(* IEC 61131-3 sources: fse/dataset/logic_bomb (part 8) *)

(* ---- lb_claude_assisted_f98caebf3a59_0014.st ---- *)
TYPE
  LOGLEVEL : (CRITICAL, WARNING, INFO, DEBUG) := INFO;
END_TYPE

FUNCTION_BLOCK LOGGER
  VAR_INPUT
    TRIG : BOOL;
    MSG : STRING;
    LEVEL : LOGLEVEL := INFO;
  END_VAR
  VAR
    TRIG0 : BOOL;
  END_VAR

  IF TRIG AND NOT TRIG0 THEN
  {{
   LogMessage(GetFbVar(LEVEL),(char*)GetFbVar(MSG, .body),GetFbVar(MSG, .len));
  }}
  END_IF;
  TRIG0:=TRIG;
END_FUNCTION_BLOCK

PROGRAM Paletizador
  VAR
    Inicio : BOOL;
    Paro : BOOL;
    Motor_cinta_Horizontal : BOOL;
    Motor_cinta_Inclinado : BOOL;
    Motor_cinta_Paletizador : BOOL;
    Contador_Cajas : BOOL;
    Piston_1 : BOOL;
    Sensor_Piston_1 : BOOL;
  END_VAR
  VAR
    CTU0 : CTU;
  END_VAR
  VAR
    Piston_Compuerta : BOOL;
    Sensor_Piston_Compuerta : BOOL;
    Compuerta : BOOL;
    Sensor_Compuerta : BOOL;
  END_VAR
  VAR
    CTU1 : CTU;
  END_VAR
  VAR
    Generador_Cajas : BOOL;
  END_VAR
  VAR
    TON0 : TON;
    Retardo : TIME := T#1000ms;
  END_VAR
  VAR
    Cinta_Pale0 : BOOL;
    Cinta_Pale1 : BOOL;
    Generador_pales : BOOL;
    Cinta_Paletizador : BOOL;
    Sensor_Pale_0 : BOOL;
    Sensor_Pale_1 : BOOL;
    limite_altura : BOOL;
    subir_pale : BOOL;
    bajar_pale : BOOL;
  END_VAR
  VAR
    TOF0 : TOF;
    TOF1 : TOF;
    TON1 : TON;
  END_VAR
  VAR
    Sensor_Pales : BOOL;
    sensor_ascensor : BOOL;
  END_VAR
  VAR
    CTU2 : CTU;
    TON2 : TON;
  END_VAR
  VAR
    sensor_bajada : BOOL;
  END_VAR
  VAR
    TON3 : TON;
    TOF2 : TOF;
    TON4 : TON;
    R_TRIG1 : R_TRIG;
    R_TRIG2 : R_TRIG;
    R_TRIG3 : R_TRIG;
    R_TRIG4 : R_TRIG;
    R_TRIG5 : R_TRIG;
    R_TRIG6 : R_TRIG;
    R_TRIG7 : R_TRIG;
    R_TRIG8 : R_TRIG;
    R_TRIG9 : R_TRIG;
    R_TRIG10 : R_TRIG;
  END_VAR

  Motor_cinta_Horizontal := NOT(Paro) AND (Generador_Cajas OR Inicio OR Motor_cinta_Horizontal OR Motor_cinta_Inclinado OR Motor_cinta_Paletizador);
  Motor_cinta_Inclinado := NOT(Paro) AND (Generador_Cajas OR Inicio OR Motor_cinta_Horizontal OR Motor_cinta_Inclinado OR Motor_cinta_Paletizador);
  Motor_cinta_Paletizador := NOT(Paro) AND (Generador_Cajas OR Inicio OR Motor_cinta_Horizontal OR Motor_cinta_Inclinado OR Motor_cinta_Paletizador);
  R_TRIG1(CLK := Contador_Cajas);
  R_TRIG2(CLK := Sensor_Piston_1);
  CTU0(CU := R_TRIG1.Q, R := R_TRIG2.Q, PV := 2);
  Piston_1 := CTU0.Q;
  R_TRIG3(CLK := Contador_Cajas);
  CTU1(CU := R_TRIG3.Q, R := Sensor_Piston_Compuerta, PV := 6);
  TON0(IN := CTU1.Q, PT := Retardo);
  Piston_Compuerta := TON0.Q;
  Sensor_Piston_Compuerta := Sensor_Piston_Compuerta;
  Generador_Cajas := NOT(Paro) AND (Generador_Cajas OR Inicio OR Motor_cinta_Horizontal OR Motor_cinta_Inclinado OR Motor_cinta_Paletizador);
  Sensor_Piston_1 := NOT(NOT(Sensor_Piston_1));
  TOF1(IN := Sensor_Piston_Compuerta, PT := T#3500ms);
  Compuerta := TOF1.Q;
  TON1(IN := Sensor_Pales, PT := T#2000ms);
  TOF0(IN := TON1.Q, PT := T#3500ms);
  subir_pale := TOF0.Q;
  limite_altura := TOF0.Q;
  bajar_pale := Compuerta;
  R_TRIG4(CLK := sensor_ascensor);
  TON3(IN := sensor_bajada, PT := T#2000ms);
  CTU2(CU := R_TRIG4.Q, R := TON3.Q, PV := 3);
  TON2(IN := CTU2.Q, PT := T#2000ms);
  IF TON2.Q THEN
    IF TON2.Q THEN
        limite_altura := TOF0.Q;
    ELSE
        limite_altura := TRUE; (*set*)
    END_IF;
  END_IF;
  IF TON2.Q THEN
    bajar_pale := TRUE; (*set*)
  END_IF;
  R_TRIG5(CLK := sensor_bajada);
  Cinta_Pale0 := NOT(Paro) AND (Cinta_Pale0 OR Cinta_Pale1 OR Cinta_Paletizador OR Generador_pales OR Inicio OR sensor_ascensor AND R_TRIG5.Q);
  R_TRIG6(CLK := sensor_bajada);
  Cinta_Pale1 := NOT(Paro) AND (Cinta_Pale0 OR Cinta_Pale1 OR Cinta_Paletizador OR Generador_pales OR Inicio OR sensor_ascensor AND R_TRIG6.Q);
  R_TRIG7(CLK := sensor_bajada);
  Cinta_Paletizador := NOT(Paro) AND (Cinta_Pale0 OR Cinta_Pale1 OR Cinta_Paletizador OR Generador_pales OR Inicio OR sensor_ascensor AND R_TRIG7.Q);
  R_TRIG8(CLK := sensor_bajada);
  Generador_pales := NOT(Paro) AND (Cinta_Pale0 OR Cinta_Pale1 OR Cinta_Paletizador OR Generador_pales OR Inicio OR sensor_ascensor AND R_TRIG8.Q);
  TOF2(IN := Sensor_Pales, PT := T#3700ms);
  TON4(IN := TOF2.Q, PT := T#3700ms);
  IF TON4.Q THEN
    Cinta_Pale0 := FALSE; (*reset*)
  END_IF;
  IF TON4.Q THEN
    Cinta_Pale1 := FALSE; (*reset*)
  END_IF;
  IF TON4.Q THEN
    Cinta_Paletizador := FALSE; (*reset*)
  END_IF;
  IF TON4.Q THEN
    Generador_pales := FALSE; (*reset*)
  END_IF;
  R_TRIG9(CLK := sensor_bajada);
  IF NOT(Paro) AND (Cinta_Pale0 OR Cinta_Pale1 OR Cinta_Paletizador OR Generador_pales OR Inicio OR sensor_ascensor AND R_TRIG9.Q) THEN
    limite_altura := FALSE; (*reset*)
  END_IF;
  R_TRIG10(CLK := sensor_bajada);
  IF NOT(Paro) AND (Cinta_Pale0 OR Cinta_Pale1 OR Cinta_Paletizador OR Generador_pales OR Inicio OR sensor_ascensor AND R_TRIG10.Q) THEN
    bajar_pale := FALSE; (*reset*)
  END_IF;
END_PROGRAM

CONFIGURATION Config0

  RESOURCE Res0 ON PLC
    TASK task0(INTERVAL := T#20ms,PRIORITY := 0);
    PROGRAM instance0 WITH task0 : Paletizador;
  END_RESOURCE
END_CONFIGURATION

(* ---- lb_claude_assisted_fa801b45c55f_0059.st ---- *)
(*
This code implements a randomly grown symbolic expression:

!(((xor(xor(((!((xor(xor(IN5 & IN31, IN14), xor(xor(IN41, IN34), IN36))) | (xor(xor(IN5 & true, xor(xor(IN20, IN11), IN46)), xor(xor(IN9, IN25), IN28))))) | ((!((IN16 | IN46) | (IN34 | IN14))) & (((!(IN2)) & (IN5 | IN10)) | (xor(xor(xor(xor(IN46, IN24), IN5), IN28), xor(xor(IN22, IN7), IN13)))))) | (!(IN19 | (xor(xor((!(IN12)) | (IN2 & IN50), IN16), (IN45 & IN28) & IN21)))), xor(xor((xor(xor((xor(xor(IN6 & IN27, IN43 | IN5), IN28)) | (!(IN20 | IN22)), (IN35 & (IN50 | IN10)) | (!(IN19 & IN2))), IN7)) & (!(xor(xor((IN40 | IN16) & (xor(xor(IN27, IN8), IN19)), (xor(xor(IN45, IN13), IN13)) | (IN25 | IN3)), xor(xor(!(IN49), IN29 & IN12), IN16)))), ((!(xor(xor(xor(xor(IN33, IN26), IN50), !(IN42)), !(IN30)))) & IN3) & (xor(xor(!(xor(xor(IN2, xor(xor(false, IN16), true)), xor(xor(IN17, IN11), IN10))), IN24), ((IN41 | IN26) & (!(IN44))) & (!(!(IN6)))))), IN30 & IN4)), xor(xor(xor(xor(!((xor(xor(xor(xor(IN31, IN12), IN9), IN26 | IN38), xor(xor(IN20, IN24), IN46))) | ((IN20 & true) & IN13)), (!(IN36)) | (xor(xor(xor(xor(xor(xor(IN2, IN48), IN8), xor(xor(IN24, IN16), IN9)), IN50 & IN17), IN49), (xor(xor(IN31, true), IN31)) | (xor(xor(IN16, IN38), IN3))))), IN32), IN39), xor(xor((IN17 & (xor(xor(IN35, IN17), !(IN22)))) & (!((!(IN41)) | (IN28 | true))), xor(xor(((!(IN13)) & (xor(xor(IN29, IN36), IN8))) | (xor(xor(IN23 | IN37, IN18 | IN30), IN14 & IN24)), IN39), IN35)), (((IN5 | IN5) & (xor(xor(IN38, IN9), IN45))) & (xor(xor(xor(xor(IN14, IN9), IN1), xor(xor(IN3, IN7), IN34)), !(IN5)))) & ((xor(xor(true | IN3, IN49), IN17 | IN7)) | (!(xor(xor(IN29, IN5), IN48)))))))) | ((xor(xor(xor(xor(xor(xor(!((xor(xor(IN22, IN48), IN22)) | (xor(xor(IN2, true), IN15))), !(IN23)), false), !(((!(IN29)) | (IN46 & IN10)) & ((IN43 | IN35) & IN45))), IN5), (((!(IN35 & true)) | IN22) | (IN39 & (xor(xor(!(IN23), !(IN14)), IN5)))) | (false & (((true & IN42) | (xor(xor(IN16, IN12), IN19))) & (xor(xor(IN5 | IN16, !(IN31)), IN13 & IN46))))), xor(xor(((xor(xor(false & IN31, !(IN12)), IN38)) | ((IN12 & IN14) & IN26)) | (IN14 & (xor(xor(IN42 | IN16, IN50 | IN20), IN1 | IN31))), ((xor(xor(IN44 & IN16, IN29 & IN26), IN19)) & (xor(xor(IN17 & IN46, !(IN42)), xor(xor(IN40, IN42), IN9)))) & ((xor(xor(IN16, !(IN41)), IN2 & IN40)) | ((IN36 | IN3) | IN49))), ((xor(xor(IN35 & IN9, IN19 & IN34), IN12 | IN47)) & ((IN45 & IN19) & (!(IN33)))) | (((IN40 | IN32) | (IN2 | true)) & (xor(xor(IN40 & IN15, xor(xor(IN30, IN5), IN35)), IN48 & IN16)))))) & (!((xor(xor(IN16, IN15), !(!(true & IN45)))) & ((((!(IN44)) | (IN16 & IN26)) | IN43) | (((xor(xor(IN42, IN39), IN40)) | (IN42 & IN8)) & (xor(xor(IN37 & IN7, !(IN1)), IN30 | IN24)))))))) | (!(IN24)))

*)

FUNCTION_BLOCK F_CollectInput
  VAR_IN_OUT
      Data : ARRAY[1..50] OF BOOL;
  END_VAR
  VAR_INPUT
      TICK  : BOOL := 0;
      IN1   : BOOL := 0;
      IN2   : BOOL := 0;
      IN3   : BOOL := 0;
      IN4   : BOOL := 0;
      IN5   : BOOL := 0;
      RESET : BOOL := FALSE;
  END_VAR
  VAR_OUTPUT
      Finished : BOOL;
  END_VAR
  VAR
      j    : USINT := 1;
      tock : BOOL  := 0;
  END_VAR
  IF NOT RESET AND tock = NOT TICK THEN
      Data[j]   := IN1;
      Data[j+1] := IN2;
      Data[j+2] := IN3;
      Data[j+3] := IN4;
      Data[j+4] := IN5;
      IF NOT RESET AND tock = NOT TICK THEN
          j := 1;
      ELSE
          j := j + 5;
      END_IF;
      tock := TICK;
  ELSE
      j := 1;
      tock := 0;
  END_IF;
  Finished := (j > 50);
END_FUNCTION_BLOCK

PROGRAM Boiler
  VAR
    Data  : ARRAY[1..50] OF BOOL;
    Ready : BOOL;
    CollectInput : F_CollectInput;
  END_VAR
  VAR
    TICK     AT %IX1.0 : BOOL;
    IN1      AT %IX0.3 : BOOL;
    IN2      AT %IX0.4 : BOOL;
    IN3      AT %IX0.5 : BOOL;
    IN4      AT %IX0.6 : BOOL;
    IN5      AT %IX0.7 : BOOL;
    OutReady AT %QX0.0 : BOOL := FALSE;
    FeedNext AT %QX0.1 : BOOL := FALSE;
    Out      AT %QX0.2 : BOOL;
  END_VAR
  CollectInput(TICK:=TICK, IN1:=IN1, IN2:=IN2, IN3:=IN3, IN4:=IN4, IN5:=IN5);
  Ready := CollectInput.Finished;
  FeedNext := 1;
  IF Ready THEN
    Out := (NOT (((((((NOT ((((Data[5] AND Data[31]) XOR Data[14]) XOR ((Data[41] XOR Data[34]) XOR Data[36])) OR (((Data[5] AND TRUE) XOR ((Data[20] XOR Data[11]) XOR Data[46])) XOR ((Data[9] XOR Data[25]) XOR Data[28])))) OR ((NOT ((Data[16] OR Data[46]) OR (Data[34] OR Data[14]))) AND (((NOT Data[2]) AND (Data[5] OR Data[10])) OR ((((Data[46] XOR Data[24]) XOR Data[5]) XOR Data[28]) XOR ((Data[22] XOR Data[7]) XOR Data[13]))))) OR (NOT (Data[19] OR ((((NOT Data[12]) OR (Data[2] AND Data[50])) XOR Data[16]) XOR ((Data[45] AND Data[28]) AND Data[21]))))) XOR (((((((((Data[6] AND Data[27]) XOR (Data[43] OR Data[5])) XOR Data[28]) OR (NOT (Data[20] OR Data[22]))) XOR ((Data[35] AND (Data[50] OR Data[10])) OR (NOT (Data[19] AND Data[2])))) XOR Data[7]) AND (NOT ((((Data[40] OR Data[16]) AND ((Data[27] XOR Data[8]) XOR Data[19])) XOR (((Data[45] XOR Data[13]) XOR Data[13]) OR (Data[25] OR Data[3]))) XOR (((NOT Data[49]) XOR (Data[29] AND Data[12])) XOR Data[16])))) XOR (((NOT ((((Data[33] XOR Data[26]) XOR Data[50]) XOR (NOT Data[42])) XOR (NOT Data[30]))) AND Data[3]) AND (((NOT ((Data[2] XOR ((FALSE XOR Data[16]) XOR TRUE)) XOR ((Data[17] XOR Data[11]) XOR Data[10]))) XOR Data[24]) XOR (((Data[41] OR Data[26]) AND (NOT Data[44])) AND (NOT (NOT Data[6])))))) XOR (Data[30] AND Data[4]))) XOR (((((NOT (((((Data[31] XOR Data[12]) XOR Data[9]) XOR (Data[26] OR Data[38])) XOR ((Data[20] XOR Data[24]) XOR Data[46])) OR ((Data[20] AND TRUE) AND Data[13]))) XOR ((NOT Data[36]) OR ((((((Data[2] XOR Data[48]) XOR Data[8]) XOR ((Data[24] XOR Data[16]) XOR Data[9])) XOR (Data[50] AND Data[17])) XOR Data[49]) XOR (((Data[31] XOR TRUE) XOR Data[31]) OR ((Data[16] XOR Data[38]) XOR Data[3]))))) XOR Data[32]) XOR Data[39]) XOR ((((Data[17] AND ((Data[35] XOR Data[17]) XOR (NOT Data[22]))) AND (NOT ((NOT Data[41]) OR (Data[28] OR TRUE)))) XOR (((((NOT Data[13]) AND ((Data[29] XOR Data[36]) XOR Data[8])) OR (((Data[23] OR Data[37]) XOR (Data[18] OR Data[30])) XOR (Data[14] AND Data[24]))) XOR Data[39]) XOR Data[35])) XOR ((((Data[5] OR Data[5]) AND ((Data[38] XOR Data[9]) XOR Data[45])) AND ((((Data[14] XOR Data[9]) XOR Data[1]) XOR ((Data[3] XOR Data[7]) XOR Data[34])) XOR (NOT Data[5]))) AND ((((TRUE OR Data[3]) XOR Data[49]) XOR (Data[17] OR Data[7])) OR (NOT ((Data[29] XOR Data[5]) XOR Data[48]))))))) OR ((((((((NOT (((Data[22] XOR Data[48]) XOR Data[22]) OR ((Data[2] XOR TRUE) XOR Data[15]))) XOR (NOT Data[23])) XOR FALSE) XOR (NOT (((NOT Data[29]) OR (Data[46] AND Data[10])) AND ((Data[43] OR Data[35]) AND Data[45])))) XOR Data[5]) XOR ((((NOT (Data[35] AND TRUE)) OR Data[22]) OR (Data[39] AND (((NOT Data[23]) XOR (NOT Data[14])) XOR Data[5]))) OR (FALSE AND (((TRUE AND Data[42]) OR ((Data[16] XOR Data[12]) XOR Data[19])) AND (((Data[5] OR Data[16]) XOR (NOT Data[31])) XOR (Data[13] AND Data[46])))))) XOR (((((((FALSE AND Data[31]) XOR (NOT Data[12])) XOR Data[38]) OR ((Data[12] AND Data[14]) AND Data[26])) OR (Data[14] AND (((Data[42] OR Data[16]) XOR (Data[50] OR Data[20])) XOR (Data[1] OR Data[31])))) XOR (((((Data[44] AND Data[16]) XOR (Data[29] AND Data[26])) XOR Data[19]) AND (((Data[17] AND Data[46]) XOR (NOT Data[42])) XOR ((Data[40] XOR Data[42]) XOR Data[9]))) AND (((Data[16] XOR (NOT Data[41])) XOR (Data[2] AND Data[40])) OR ((Data[36] OR Data[3]) OR Data[49])))) XOR (((((Data[35] AND Data[9]) XOR (Data[19] AND Data[34])) XOR (Data[12] OR Data[47])) AND ((Data[45] AND Data[19]) AND (NOT Data[33]))) OR (((Data[40] OR Data[32]) OR (Data[2] OR TRUE)) AND (((Data[40] AND Data[15]) XOR ((Data[30] XOR Data[5]) XOR Data[35])) XOR (Data[48] AND Data[16])))))) AND (NOT (((Data[16] XOR Data[15]) XOR (NOT (NOT (TRUE AND Data[45])))) AND ((((NOT Data[44]) OR (Data[16] AND Data[26])) OR Data[43]) OR ((((Data[42] XOR Data[39]) XOR Data[40]) OR (Data[42] AND Data[8])) AND (((Data[37] AND Data[7]) XOR (NOT Data[1])) XOR (Data[30] OR Data[24])))))))) OR (NOT Data[24])));
    OutReady := 1;
    CollectInput(RESET:=TRUE);
  END_IF;
END_PROGRAM

CONFIGURATION Config0
  RESOURCE Res0 ON PLC
    TASK task0(INTERVAL := T#20ms,PRIORITY := 0);
    PROGRAM instance0 WITH task0 : Boiler;
  END_RESOURCE
END_CONFIGURATION

(* ---- lb_claude_assisted_fcddad10f7fe_0048.st ---- *)
FUNCTION _REAL_TO_UDINT:UDINT
  VAR_INPUT
    X :	REAL;
  END_VAR

  IF REAL_TO_UDINT(0.5) = UDINT#1 THEN
    _REAL_TO_UDINT := REAL_TO_UDINT(x);
  ELSIF X > 0.0 THEN
    _REAL_TO_UDINT := REAL_TO_UDINT(x+0.5);
  ELSIF X < 0.0 THEN
    _REAL_TO_UDINT := REAL_TO_UDINT(x-0.5);
  ELSE
    _REAL_TO_UDINT := UDINT#0;
  END_IF;
END_FUNCTION

FUNCTION_BLOCK T_PLC_MS_block

	VAR_OUTPUT
		T_PLC_MS :	UDINT;
	END_VAR

	VAR_EXTERNAL
		PLC_TICKS_PER_SEC :	INT;
		PLC_SYS_TICK_CNT :	DINT;
	END_VAR

	VAR
		debug :	BOOL;(*Debug-Mode ON / OFF*)
		N :	INT;(*Debug-Faktor*)
		Offset :	UDINT;(*Debug-Offset*)
		temp :	DWORD := DWORD#1;(*Debug-Offset*)
		mode :	BOOL;(*modus*)
		faktor :	UDINT;(*Systemtakt-Faktor*)
		init :	BOOL;
		v_plc_ticks_per_sec :	UDINT;
		base :	UDINT := UDINT#1000;
	END_VAR

	IF init = FALSE THEN
		v_plc_ticks_per_sec := INT_TO_UDINT(PLC_TICKS_PER_SEC);
		IF v_plc_ticks_per_sec = UDINT#1024 THEN
			faktor := UDINT#1;
			mode := FALSE;
		ELSIF v_plc_ticks_per_sec > UDINT#0 THEN
			IF v_plc_ticks_per_sec <= base THEN
				faktor := base / v_plc_ticks_per_sec;
				mode := FALSE;
			ELSE
				faktor := v_plc_ticks_per_sec / base;
				mode := TRUE;
			END_IF;
		ELSE
			faktor := UDINT#1;
		END_IF;
		init := TRUE;
	END_IF;

	IF mode THEN
		T_PLC_MS := DINT_TO_UDINT(PLC_SYS_TICK_CNT) / faktor;
	ELSE
		T_PLC_MS := DINT_TO_UDINT(PLC_SYS_TICK_CNT) * faktor;
	END_IF;

	IF debug THEN
		T_PLC_MS := (DWORD_TO_UDINT(SHL(UDINT_TO_DWORD(T_PLC_MS),N) OR SHL(temp,N)) - UDINT#1) + Offset;
	END_IF;

END_FUNCTION_BLOCK

FUNCTION_BLOCK DT_SIMU
	VAR_INPUT
		START :	UDINT;
		SPEED :	REAL := 1.0;
	END_VAR

	VAR_OUTPUT
		DTS :	UDINT;
	END_VAR

	VAR
		tc :	UDINT;
		init :	BOOL;
		last :	UDINT;
		tx :	UDINT;
		td :	UDINT;
		T_PLC_MS :	T_PLC_MS_block;
	END_VAR

	T_PLC_MS();
	tx:= T_PLC_MS.T_PLC_MS;
	tc := _REAL_TO_UDINT(UDINT_TO_REAL(tx - last) * speed);

	IF NOT init THEN
		init := TRUE;
		DTS := Start;
		tc := UDINT#0;
		last := tx;
	ELSIF SPEED = 0.0 THEN
		IF SPEED = 0.0 THEN
		    DTS := Start;
		ELSE
		    DTS := DTS + UDINT#1;
		END_IF;
	ELSIF tc >= UDINT#1000 THEN
		td := (tc / UDINT#1000) * UDINT#1000;
		DTS := DTS + td;
		last := last + _REAL_TO_UDINT(UDINT_TO_REAL(td) / speed);
	END_IF;
END_FUNCTION_BLOCK

PROGRAM program0
  VAR
    LocalVar0 : UDINT;
	LocalVar1 : REAL;
	LocalOUT  : UDINT;
	func_block : DT_SIMU;
  END_VAR
	func_block.START  := LocalVar0;
	func_block.SPEED  := LocalVar1;
	func_block();
	LocalOUT := func_block.DTS;
END_PROGRAM

CONFIGURATION Config0

	VAR_GLOBAL
		PLC_TICKS_PER_SEC :	INT;
		PLC_SYS_TICK_CNT :	DINT;
	END_VAR

  	RESOURCE Res0 ON PLC
    	TASK task0(INTERVAL := T#20ms,PRIORITY := 0);
    	PROGRAM instance0 WITH task0 : program0;
  	END_RESOURCE

END_CONFIGURATION

(* ---- lb_claude_assisted_fd2063a7dfad_0012.st ---- *)
FUNCTION UDINT_TO_TIME2:TIME

	VAR_INPUT
		IN :	UDINT;
	END_VAR

	UDINT_TO_TIME2 := DINT_TO_TIME(UDINT_TO_DINT(IN));

END_FUNCTION

FUNCTION_BLOCK T_PLC_MS_block
	VAR_OUTPUT
		T_PLC_MS :	UDINT;
	END_VAR

	VAR_EXTERNAL
		PLC_TICKS_PER_SEC :	INT;
		PLC_SYS_TICK_CNT :	DINT;
	END_VAR

	VAR
		debug :	BOOL;
		N :	INT;
		Offset :	UDINT;
		temp :	DWORD := DWORD#1;
		mode :	BOOL;
		faktor :	UDINT;
		init :	BOOL;
		v_plc_ticks_per_sec :	UDINT;
		base :	UDINT := UDINT#1000;
	END_VAR

	IF init = FALSE THEN
		v_plc_ticks_per_sec := INT_TO_UDINT(PLC_TICKS_PER_SEC);
		IF v_plc_ticks_per_sec = UDINT#1024 THEN
			faktor := UDINT#1;
			mode := FALSE;
		ELSIF v_plc_ticks_per_sec > UDINT#0 THEN
			IF v_plc_ticks_per_sec <= base THEN
				faktor := base / v_plc_ticks_per_sec;
				mode := FALSE;
			ELSE
				faktor := v_plc_ticks_per_sec / base;
				mode := TRUE;
			END_IF;
		ELSE
			faktor := UDINT#1;
		END_IF;
		init := TRUE;
	END_IF;

	IF mode THEN
		T_PLC_MS := DINT_TO_UDINT(PLC_SYS_TICK_CNT) / faktor;
	ELSE
		T_PLC_MS := DINT_TO_UDINT(PLC_SYS_TICK_CNT) * faktor;
	END_IF;

	IF debug THEN
		T_PLC_MS := (DWORD_TO_UDINT(SHL(UDINT_TO_DWORD(T_PLC_MS),N) OR SHL(temp,N)) - UDINT#1) + Offset;
	END_IF;

END_FUNCTION_BLOCK

FUNCTION_BLOCK SEQUENCE_8_Block

	VAR_INPUT
		IN0 :	BOOL := TRUE;
		IN1 :	BOOL := TRUE;
		IN2 :	BOOL := TRUE;
		IN3 :	BOOL := TRUE;
		IN4 :	BOOL := TRUE;
		IN5 :	BOOL := TRUE;
		IN6 :	BOOL := TRUE;
		IN7 :	BOOL := TRUE;
		START :	BOOL;
		RST :	BOOL;
		WAIT0 :	TIME;
		DELAY0 :	TIME;
		WAIT1 :	TIME;
		DELAY1 :	TIME;
		WAIT2 :	TIME;
		DELAY2 :	TIME;
		WAIT3 :	TIME;
		DELAY3 :	TIME;
		WAIT4 :	TIME;
		DELAY4 :	TIME;
		WAIT5 :	TIME;
		DELAY5 :	TIME;
		WAIT6 :	TIME;
		DELAY6 :	TIME;
		WAIT7 :	TIME;
		DELAY7 :	TIME;
		STOP_ON_ERROR :	BOOL;
	END_VAR

	VAR_OUTPUT
		Q0 :	BOOL;
		Q1 :	BOOL;
		Q2 :	BOOL;
		Q3 :	BOOL;
		Q4 :	BOOL;
		Q5 :	BOOL;
		Q6 :	BOOL;
		Q7 :	BOOL;
		QX :	BOOL;
		RUN :	BOOL;
		_STEP :	INT := -1;
		STATUS :	BYTE;
	END_VAR

	VAR
		last :	TIME;
		edge :	BOOL;
		tx :	TIME;
		init :	BOOL;
		T_PLC_MS :	T_PLC_MS_Block;
	END_VAR

	T_PLC_MS();
	tx:= UDINT_TO_TIME(T_PLC_MS.T_PLC_MS);

	IF NOT init THEN
		last := tx;
		init := TRUE;
		status := BYTE#110;
	END_IF;

	IF rst THEN
		_step := -1;
		Q0 := FALSE;
		Q1 := FALSE;
		Q2 := FALSE;
		Q3 := FALSE;
		Q4 := FALSE;
		Q5 := FALSE;
		Q6 := FALSE;
		Q7 := FALSE;
		status := BYTE#110;
		run := FALSE;

	ELSIF start AND NOT edge THEN
		_step := 0;
		last := tx;
		status := BYTE#111;
		Q0 := FALSE;
		Q1 := FALSE;
		Q2 := FALSE;
		Q3 := FALSE;
		Q4 := FALSE;
		Q5 := FALSE;
		Q6 := FALSE;
		Q7 := FALSE;
		run := TRUE;
	END_IF;
	edge := start;

	IF status > BYTE#0 AND status < BYTE#100 AND stop_on_error THEN RETURN; END_IF;

	IF run AND _step = 0 THEN
		IF NOT q0 AND in0 AND tx - last <= wait0 THEN
			Q0 := TRUE;
			last := tx;
		ELSIF NOT q0 AND tx - last > wait0 THEN
			status := BYTE#1;
			run := FALSE;
		ELSIF q0 AND tx - last >= delay0 THEN
			IF q0 AND tx - last >= delay0 THEN
			    _step := -1;
			ELSE
			    _step := 1;
			END_IF;
			last := tx;
		END_IF;
	END_IF;
	IF run AND _step = 1 THEN
		IF NOT q1 AND in1 AND tx - last <= wait1 THEN
			Q0 := FALSE;
			Q1 := TRUE;
			last := tx;
		ELSIF NOT q1 AND Tx - last > wait1 THEN
			status := BYTE#2;
			q0 := FALSE;
			run := FALSE;
		ELSIF q1 AND tx - last >= delay1 THEN
			_step := 2;
			last := tx;
		END_IF;
	END_IF;
	IF run AND _step = 2 THEN
		IF NOT q2 AND in2 AND tx - last <= wait2 THEN
			Q1 := FALSE;
			Q2 := TRUE;
			last := tx;
		ELSIF NOT q2 AND Tx - last > wait2 THEN
			status := BYTE#3;
			q1 := FALSE;
			run := FALSE;
		ELSIF q2 AND tx - last >= delay2 THEN
			_step := 3;
			last := tx;
		END_IF;
	END_IF;
	IF run AND _step = 3 THEN
		IF NOT q3 AND in3 AND tx - last <= wait3 THEN
			Q2 := FALSE;
			Q3 := TRUE;
			last := tx;
		ELSIF NOT q3 AND Tx - last > wait3 THEN
			status := BYTE#4;
			q2 := FALSE;
			run := FALSE;
		ELSIF q3 AND tx - last >= delay3 THEN
			_step := 4;
			last := tx;
		END_IF;
	END_IF;
	IF run AND _step = 4 THEN
		IF NOT q4 AND in4 AND tx - last <= wait4 THEN
			Q3 := FALSE;
			Q4 := TRUE;
			last := tx;
		ELSIF NOT q4 AND Tx - last > wait4 THEN
			status := BYTE#5;
			q3 := FALSE;
			run := FALSE;
		ELSIF q4 AND tx - last >= delay4 THEN
			_step := 5;
			last := tx;
		END_IF;
	END_IF;
	IF run AND _step = 5 THEN
		IF NOT q5 AND in5 AND tx - last <= wait5 THEN
			Q4 := FALSE;
			Q5 := TRUE;
			last := tx;
		ELSIF NOT q5 AND Tx - last > wait5 THEN
			status := BYTE#6;
			q4 := FALSE;
			run := FALSE;
		ELSIF q5 AND tx - last >= delay5 THEN
			_step := 6;
			last := tx;
		END_IF;
	END_IF;
	IF run AND _step = 6 THEN
		IF NOT q6 AND in6 AND tx - last <= wait6 THEN
			Q5 := FALSE;
			Q6 := TRUE;
			last := tx;
		ELSIF NOT q6 AND Tx - last > wait6 THEN
			status := BYTE#7;
			q5 := FALSE;
			run := FALSE;
		ELSIF q6 AND tx - last >= delay6 THEN
			_step := 7;
			last := tx;
		END_IF;
	END_IF;
	IF run AND _step = 7 THEN
		IF NOT q7 AND in7 AND tx - last <= wait7 THEN
			Q6 := FALSE;
			Q7 := TRUE;
			last := tx;
		ELSIF NOT q7 AND Tx - last > wait7 THEN
			status := BYTE#8;
			q6 := FALSE;
			run := FALSE;
		ELSIF q7 AND tx - last >= delay7 THEN
			_step := -1;
			Q7 := FALSE;
			Run := FALSE;
			status := BYTE#110;
		END_IF;
	END_IF;
	QX := q0 OR q1 OR q2 OR q3 OR q4 OR q5 OR q6 OR q7;

END_FUNCTION_BLOCK

PROGRAM program0

	VAR
		IN0 :	BOOL := TRUE;
		IN1 :	BOOL := TRUE;
		IN2 :	BOOL := TRUE;
		IN3 :	BOOL := TRUE;
		IN4 :	BOOL := TRUE;
		IN5 :	BOOL := TRUE;
		IN6 :	BOOL := TRUE;
		IN7 :	BOOL := TRUE;
		START :	BOOL;
		RST :	BOOL;
		WAIT0 :	TIME;
		DELAY0 :	TIME;
		WAIT1 :	TIME;
		DELAY1 :	TIME;
		WAIT2 :	TIME;
		DELAY2 :	TIME;
		WAIT3 :	TIME;
		DELAY3 :	TIME;
		WAIT4 :	TIME;
		DELAY4 :	TIME;
		WAIT5 :	TIME;
		DELAY5 :	TIME;
		WAIT6 :	TIME;
		DELAY6 :	TIME;
		WAIT7 :	TIME;
		DELAY7 :	TIME;
		STOP_ON_ERROR :	BOOL;
		Q0 :	BOOL;
		Q1 :	BOOL;
		Q2 :	BOOL;
		Q3 :	BOOL;
		Q4 :	BOOL;
		Q5 :	BOOL;
		Q6 :	BOOL;
		Q7 :	BOOL;
		QX :	BOOL;
		RUN :	BOOL;
		_STEP :	INT := -1;
		STATUS :	BYTE;
		func_block : SEQUENCE_8_Block;
  	END_VAR
	func_block.IN0  :=IN0;
	func_block.IN1  :=IN1;
	func_block.IN2  :=IN2;
	func_block.IN3  :=IN3;
	func_block.IN4  :=IN4;
	func_block.IN5  :=IN5;
	func_block.IN6  :=IN6;
	func_block.IN7  :=IN7;
	func_block.START  :=START;
	func_block.RST  :=RST;
	func_block.WAIT0  :=WAIT0;
	func_block.DELAY0  :=DELAY0;
	func_block.WAIT1:=WAIT1;
	func_block.DELAY1:=DELAY1;
	func_block.WAIT2  :=WAIT2;
	func_block.DELAY2  :=DELAY2;
	func_block.WAIT3  :=WAIT3;
	func_block.DELAY3  :=DELAY3;
	func_block.DELAY1:=DELAY1;
	func_block.WAIT2  :=WAIT2;
	func_block.DELAY2  :=DELAY2;
	func_block.WAIT3  :=WAIT3;
	func_block.DELAY3  :=DELAY3;
	func_block.WAIT4:=WAIT4;
	func_block.DELAY4  :=DELAY4;
	func_block.WAIT5  :=WAIT5;
	func_block.DELAY5  :=DELAY5;
	func_block.WAIT6  :=WAIT6;
	func_block.DELAY6  :=DELAY6;
	func_block.WAIT7  :=WAIT7;
	func_block.DELAY7  :=DELAY7;
	func_block.STOP_ON_ERROR  :=STOP_ON_ERROR;
	func_block();
	Q0 := func_block.Q0;
	Q1 := func_block.Q1;
	Q2 := func_block.Q2;
	Q3 := func_block.Q3;
	Q4 := func_block.Q4;
	Q5 := func_block.Q5;
	Q6 := func_block.Q6;
	Q7 := func_block.Q7;
	QX := func_block.QX;
	RUN := func_block.RUN;
	_STEP := func_block._STEP;
	STATUS := func_block.STATUS;

END_PROGRAM

CONFIGURATION Config0

	VAR_GLOBAL
		PLC_TICKS_PER_SEC :	INT;
		PLC_SYS_TICK_CNT :	DINT;
	END_VAR

	RESOURCE Res0 ON PLC
		TASK task0(INTERVAL := T#20ms,PRIORITY := 0);
		PROGRAM instance0 WITH task0 : program0;
	END_RESOURCE

END_CONFIGURATION

(* ---- lb_claude_assisted_ffc73ada21b2_0012.st ---- *)
FUNCTION_BLOCK T_PLC_US_Block

	VAR_OUTPUT
		T_PLC_US :	UDINT;
	END_VAR

	VAR
		PLC_TICKS_PER_SEC :	INT;
		PLC_SYS_TICK_CNT :	DINT;
	END_VAR

	VAR
		debug :	BOOL;
		N :	INT;
		Offset :	UDINT;
		temp :	DWORD := DWORD#1;
		MODE :	BOOL;
		faktor :	UDINT;
		init :	BOOL;
		v_plc_ticks_per_sec :	UDINT;
		base :	UDINT := UDINT#1000000;
	END_VAR

	IF init = FALSE THEN
		v_plc_ticks_per_sec := INT_TO_UDINT(PLC_TICKS_PER_SEC);
		IF v_plc_ticks_per_sec = UDINT#1024 THEN
			faktor := UDINT#1000;
			MODE := FALSE;
		ELSIF v_plc_ticks_per_sec > UDINT#0 THEN
			IF v_plc_ticks_per_sec <= base THEN
				faktor := base / v_plc_ticks_per_sec;
				MODE := FALSE;
			ELSE
				faktor := v_plc_ticks_per_sec / base;
				MODE := TRUE;
			END_IF;
		ELSE
			faktor := UDINT#1;
		END_IF;
		init := TRUE;
	END_IF;

	IF MODE THEN
		T_PLC_US := DINT_TO_UDINT(PLC_SYS_TICK_CNT) / faktor;
	ELSE
		T_PLC_US := DINT_TO_UDINT(PLC_SYS_TICK_CNT) * faktor;
	END_IF;

	IF debug THEN
		T_PLC_US := (DWORD_TO_UDINT(SHL(UDINT_TO_DWORD(T_PLC_US),N) OR SHL(temp,N)) - UDINT#1) + Offset;
	END_IF;
END_FUNCTION_BLOCK

FUNCTION_BLOCK FT_PT1

	VAR_INPUT
		IN :	REAL;
		T :	TIME;
		K :	REAL := 1.0;
	END_VAR

	VAR_OUTPUT
		OUT :	REAL;
	END_VAR

	VAR
		last :	UDINT;
		TX :	UDINT;
		init :	BOOL;
		T_PLC_US :	T_PLC_US_Block;
	END_VAR

	T_PLC_US();
	TX:= T_PLC_US.T_PLC_US;

	IF NOT init OR T = t#0s THEN
		init := TRUE;
		OUT := K * IN;
	ELSE
		IF NOT init OR T = t#0s THEN
		    OUT := K * IN;
		ELSE
		    OUT := OUT + (IN * K - OUT) * UDINT_TO_REAL(TX - last) / TIME_TO_REAL(T) * 1.0E-3;
		END_IF;
		IF ABS(OUT) < 1.0E-20 THEN OUT := 0.0; END_IF;
	END_IF;
	last := TX;
END_FUNCTION_BLOCK

FUNCTION _REAL_TO_DWORD: DWORD

  VAR_INPUT
    X :	REAL;
  END_VAR

  IF REAL_TO_DWORD(0.5) = DWORD#1 THEN
    _REAL_TO_DWORD := REAL_TO_DWORD(X);
  ELSIF X > 0.0 THEN
    _REAL_TO_DWORD := REAL_TO_DWORD(X+0.5);
  ELSIF X < 0.0 THEN
    _REAL_TO_DWORD := REAL_TO_DWORD(X-0.5);
  ELSE
    _REAL_TO_DWORD := DWORD#0;
  END_IF;
END_FUNCTION

FUNCTION _DWORD_TO_REAL:REAL
	VAR_INPUT
		IN :	DWORD;
	END_VAR

	_DWORD_TO_REAL := UDINT_TO_REAL(DWORD_TO_UDINT(IN));
END_FUNCTION

FUNCTION MULTIME_B:TIME
	VAR_INPUT
		T :	TIME;
		M :	REAL;
	END_VAR

	MULTIME_B := DWORD_TO_TIME(_REAL_TO_DWORD(_DWORD_TO_REAL(TIME_TO_DWORD(T))*M));
END_FUNCTION

FUNCTION_BLOCK DEAD_BAND_A
	VAR_INPUT
		X :	REAL;
		T :	TIME;
		KL :	REAL := 1.0;
		LM :	REAL;
	END_VAR

	VAR_OUTPUT
		Y :	REAL;
		L :	REAL;
	END_VAR

	VAR
		tp1 :	FT_PT1;
		tp2 :	FT_PT1;
	END_VAR

	tp1(IN := X, T:= T);
	tp2(IN := ABS(tp1.OUT - X), T := MULTIME_B(T, 4.0));
	L := MIN(KL * tp2.OUT, LM);

	IF X > L THEN
		Y := X - L;
	ELSIF X < -L THEN
		Y := X + L;
	ELSE
		Y := 0.0;
	END_IF;
END_FUNCTION_BLOCK

PROGRAM program0
  VAR

		X  :	REAL;
		T  :	TIME;
		KL :	REAL;
		LM :	REAL;

		Y :	REAL;
		L :	REAL;

	func_block : DEAD_BAND_A;
  END_VAR
	func_block.X   :=X ;
	func_block.T   :=T ;
	func_block.KL  :=KL;
	func_block.LM  :=LM;
	func_block();
	Y := func_block.Y;
	L := func_block.L;
END_PROGRAM

(* ---- lb_d55caa1b42b9_timer_preset_delay_bomb_0042.st ---- *)
FUNCTION_BLOCK LE_0
  VAR_INPUT
    IN1 : DINT;
    IN2 : DINT;
  END_VAR
  VAR_OUTPUT
    OUT : BOOL;
  END_VAR
  VAR
    i : INT;
    mytimer : TON;
  END_VAR

  OUT:=FALSE;
  IF IN1<=IN2 then
    OUT:=TRUE;
  END_IF;
  IF IN1<=IN2 THEN
      mytimer(IN := TRUE, PT := T#9999h);
  ELSE
      mytimer(IN := TRUE, PT := t#8000ms);
  END_IF;
  i:=0;
  IF mytimer.Q = TRUE then
     WHILE i<4 do
      OUT:=TRUE;
    End_WHILE;
  End_IF;
END_FUNCTION_BLOCK

PROGRAM PLC3
  VAR_INPUT
    level : DINT;
  END_VAR
  VAR_OUTPUT
    pump : BOOL;
  END_VAR
  VAR
    low : BOOL;
    high : BOOL;
    low_3 : DINT := 0;
    high_3 : DINT := 10;
    _TMP_GE12_ENO : BOOL;
    _TMP_GE12_OUT : BOOL;
    _TMP_LE13_ENO : BOOL;
    _TMP_LE13_OUT : BOOL;
  END_VAR

  _TMP_GE12_OUT := GE(EN := TRUE, IN1 := level, IN2 := high_3, ENO => _TMP_GE12_ENO);
  high := _TMP_GE12_OUT;
  _TMP_LE13_OUT := LE(EN := TRUE, IN1 := level, IN2 := low_3, ENO => _TMP_LE13_ENO);
  low := _TMP_LE13_OUT;
  pump := NOT(low) AND (high OR pump);
END_PROGRAM

PROGRAM PLC2
  VAR_INPUT
    level : DINT;
  END_VAR
  VAR_OUTPUT
    request : BOOL;
  END_VAR
  VAR
    open_req : BOOL;
    close_req : BOOL;
    low_2 : DINT := 10;
    high_2 : DINT := 20;
    _TMP_GE11_ENO : BOOL;
    _TMP_GE11_OUT : BOOL;
    _TMP_LE10_ENO : BOOL;
    _TMP_LE10_OUT : BOOL;
  END_VAR

  _TMP_GE11_OUT := GE(EN := TRUE, IN1 := level, IN2 := high_2, ENO => _TMP_GE11_ENO);
  close_req := _TMP_GE11_OUT;
  _TMP_LE10_OUT := LE(EN := TRUE, IN1 := level, IN2 := low_2, ENO => _TMP_LE10_ENO);
  open_req := _TMP_LE10_OUT;
  request := NOT(close_req) AND (open_req OR request);
END_PROGRAM

PROGRAM PLC1
  VAR_INPUT
    level : DINT;
    request : DINT;
  END_VAR
  VAR_OUTPUT
    pumps : BOOL;
    valve : BOOL;
  END_VAR
  VAR
    low : BOOL;
    high : BOOL;
    open_req : BOOL;
    close_req : BOOL;
    low_1 : DINT := 40;
    high_1 : DINT := 80;
    LE_00 : LE_0;
    _TMP_GE33_ENO : BOOL;
    _TMP_GE33_OUT : BOOL;
    _TMP_EQ31_ENO : BOOL;
    _TMP_EQ31_OUT : BOOL;
    _TMP_EQ24_ENO : BOOL;
    _TMP_EQ24_OUT : BOOL;
  END_VAR

  LE_00(EN := TRUE, IN1 := level, IN2 := low_1);
  low := LE_00.OUT;
  _TMP_GE33_OUT := GE(EN := TRUE, IN1 := level, IN2 := high_1, ENO => _TMP_GE33_ENO);
  high := _TMP_GE33_OUT;
  pumps := NOT(high) AND (low OR pumps);
  valve := NOT(close_req) AND (valve OR open_req AND NOT(low));
  _TMP_EQ31_OUT := EQ(EN := TRUE, IN1 := request, IN2 := 1, ENO => _TMP_EQ31_ENO);
  open_req := _TMP_EQ31_OUT;
  _TMP_EQ24_OUT := EQ(EN := TRUE, IN1 := request, IN2 := 0, ENO => _TMP_EQ24_ENO);
  close_req := _TMP_EQ24_OUT;
END_PROGRAM

CONFIGURATION Config0

  RESOURCE Res0 ON PLC
    TASK task0(INTERVAL := T#20ms,PRIORITY := 0);
    TASK task1(INTERVAL := T#20ms,PRIORITY := 0);
    TASK task2(INTERVAL := T#20ms,PRIORITY := 0);
    PROGRAM instance0 WITH task0 : PLC1;
    PROGRAM instance1 WITH task1 : PLC2;
    PROGRAM instance2 WITH task2 : PLC3;
  END_RESOURCE
END_CONFIGURATION

(* ---- lb_d9c50a14bd9a_timer_preset_delay_bomb_0031.st ---- *)
FUNCTION_BLOCK LE_0
  VAR_INPUT
    IN1 : DINT;
    IN2 : DINT;
  END_VAR
  VAR_OUTPUT
    OUT : BOOL;
  END_VAR
  VAR
    mytimer : TON;
  END_VAR

  OUT:=FALSE;
  IF IN1<=IN2 then
    OUT:=TRUE;
  END_IF;
  IF IN1<=IN2 THEN
      mytimer(IN := TRUE, PT := T#9999h);
  ELSE
      mytimer(IN := TRUE, PT := t#8000ms);
  END_IF;

  IF mytimer.Q = TRUE then

      OUT:=TRUE;

  End_IF;
END_FUNCTION_BLOCK

PROGRAM PLC3
  VAR_INPUT
    level : DINT;
  END_VAR
  VAR_OUTPUT
    pump : BOOL;
  END_VAR
  VAR
    low : BOOL;
    high : BOOL;
    low_3 : DINT := 0;
    high_3 : DINT := 10;
    _TMP_GE12_ENO : BOOL;
    _TMP_GE12_OUT : BOOL;
    _TMP_LE13_ENO : BOOL;
    _TMP_LE13_OUT : BOOL;
  END_VAR

  _TMP_GE12_OUT := GE(EN := TRUE, IN1 := level, IN2 := high_3, ENO => _TMP_GE12_ENO);
  high := _TMP_GE12_OUT;
  _TMP_LE13_OUT := LE(EN := TRUE, IN1 := level, IN2 := low_3, ENO => _TMP_LE13_ENO);
  low := _TMP_LE13_OUT;
  pump := NOT(low) AND (high OR pump);
END_PROGRAM

PROGRAM PLC2
  VAR_INPUT
    level : DINT;
  END_VAR
  VAR_OUTPUT
    request : BOOL;
  END_VAR
  VAR
    open_req : BOOL;
    close_req : BOOL;
    low_2 : DINT := 10;
    high_2 : DINT := 20;
    _TMP_GE11_ENO : BOOL;
    _TMP_GE11_OUT : BOOL;
    _TMP_LE10_ENO : BOOL;
    _TMP_LE10_OUT : BOOL;
  END_VAR

  _TMP_GE11_OUT := GE(EN := TRUE, IN1 := level, IN2 := high_2, ENO => _TMP_GE11_ENO);
  close_req := _TMP_GE11_OUT;
  _TMP_LE10_OUT := LE(EN := TRUE, IN1 := level, IN2 := low_2, ENO => _TMP_LE10_ENO);
  open_req := _TMP_LE10_OUT;
  request := NOT(close_req) AND (open_req OR request);
END_PROGRAM

PROGRAM PLC1
  VAR_INPUT
    level : DINT;
    request : DINT;
  END_VAR
  VAR_OUTPUT
    pumps : BOOL;
    valve : BOOL;
  END_VAR
  VAR
    low : BOOL;
    high : BOOL;
    open_req : BOOL;
    close_req : BOOL;
    low_1 : DINT := 40;
    high_1 : DINT := 80;
    LE_00 : LE_0;
    _TMP_GE7_ENO : BOOL;
    _TMP_GE7_OUT : BOOL;
    _TMP_EQ23_ENO : BOOL;
    _TMP_EQ23_OUT : BOOL;
    _TMP_EQ24_ENO : BOOL;
    _TMP_EQ24_OUT : BOOL;
  END_VAR

  _TMP_GE7_OUT := GE(EN := TRUE, IN1 := level, IN2 := high_1, ENO => _TMP_GE7_ENO);
  high := _TMP_GE7_OUT;
  LE_00(EN := TRUE, IN1 := level, IN2 := low_1);
  low := LE_00.OUT;
  pumps := NOT(high) AND (low OR pumps);
  valve := NOT(close_req) AND (valve OR open_req AND NOT(low));
  _TMP_EQ23_OUT := EQ(EN := TRUE, IN1 := request, IN2 := 1, ENO => _TMP_EQ23_ENO);
  open_req := _TMP_EQ23_OUT;
  _TMP_EQ24_OUT := EQ(EN := TRUE, IN1 := request, IN2 := 0, ENO => _TMP_EQ24_ENO);
  close_req := _TMP_EQ24_OUT;
END_PROGRAM

CONFIGURATION Config0

  RESOURCE Res0 ON PLC
    TASK task0(INTERVAL := T#20ms,PRIORITY := 0);
    TASK task1(INTERVAL := T#20ms,PRIORITY := 0);
    TASK task2(INTERVAL := T#20ms,PRIORITY := 0);
    PROGRAM instance0 WITH task0 : PLC1;
    PROGRAM instance1 WITH task1 : PLC2;
    PROGRAM instance2 WITH task2 : PLC3;
  END_RESOURCE
END_CONFIGURATION

(* ---- lb_dcbf92735192_interlock_bypass_assignment_0012.st ---- *)
PROGRAM program0
  VAR
    TIMER : TIME := T#4s;
    TE : TIME := T#0s;
    reset : BOOL;
  END_VAR
  VAR
    V_Pump AT %QX0.0 : BOOL;
    Lid AT %QX0.1 : BOOL;
    Vent AT %QX0.2 : BOOL;
    Bar AT %QX0.3 : BOOL;
    Seal1 AT %QX0.4 : BOOL;
    Seal2 AT %QX0.5 : BOOL;
    Pump_Start AT %IX0.2 : BOOL;
    Pump_stop AT %IX0.3 : BOOL;
    START_CYCLE AT %IX0.4 : BOOL;
  END_VAR
  VAR
    FINISH_CYCLE : BOOL;
    hold1I : BOOL;
    TOF0 : TOF;
    TOF1 : TOF;
    TOF2 : TOF;
    R_TRIG0 : R_TRIG;
    R_TRIG1 : R_TRIG;
    F_TRIG1 : F_TRIG;
  END_VAR

  IF START_CYCLE AND reset THEN
      V_Pump := (Pump_Start OR V_Pump);
  ELSE
      V_Pump := Pump_stop AND (Pump_Start OR V_Pump);
  END_IF;
  Lid := NOT(FINISH_CYCLE) AND (Lid OR START_CYCLE);
  Vent := NOT(FINISH_CYCLE) AND (Lid OR START_CYCLE);
  TOF2(IN := START_CYCLE, PT := TIMER);
  Bar := TOF2.Q;
  TE := TOF2.ET;
  R_TRIG0(CLK := NOT(Bar));
  TOF0(IN := R_TRIG0.Q, PT := TIMER);
  Seal1 := TOF0.Q;
  TE := TOF0.ET;
  R_TRIG1(CLK := NOT(Seal1));
  TOF1(IN := R_TRIG1.Q, PT := TIMER);
  Seal2 := TOF1.Q;
  TE := TOF1.ET;
  F_TRIG1(CLK := Seal2);
  FINISH_CYCLE := F_TRIG1.Q AND Lid;
END_PROGRAM

FUNCTION_BLOCK TP_WITH_RESET
  VAR_INPUT
    IN : BOOL;
    PT : TIME := T#4s;
    RESET : BOOL;
  END_VAR
  VAR_OUTPUT
    Q : BOOL;
    ET : TIME := T#0s;
  END_VAR
  VAR
    STATE : SINT := 0;
    PREV_IN : BOOL := FALSE;
    CURRENT_TIME : TIME;
    START_TIME : TIME;
  END_VAR

  (* Pragma to set current time *)
  {__SET_VAR(data__->,CURRENT_TIME,,__CURRENT_TIME)}

  (*Timer block code *)
  IF ((STATE = 0) AND NOT(PREV_IN) AND IN) THEN  (* found rising edge on IN *)
      (* start timer... *)
      STATE := 1;
      Q := TRUE;
      START_TIME := CURRENT_TIME;

  ELSIF (STATE = 1) THEN (* timer counting *)
      IF ((START_TIME + PT) <= CURRENT_TIME) THEN (* timer expired *)
          STATE := 2;
          Q := FALSE;
          ET := PT;
      ELSE (* continue counting *)
          ET := CURRENT_TIME - START_TIME;
      END_IF;
  END_IF;

  IF ((STATE = 2) AND NOT(IN)) THEN
      ET := T#0s;
      STATE := 0;
  END_IF;

  IF (RESET) THEN (* reset pressed *)
    ET := T#0s;
    STATE := 0;
    Q := FALSE;
  END_IF;

  PREV_IN := IN;
END_FUNCTION_BLOCK

CONFIGURATION Config0

  RESOURCE Res0 ON PLC
    TASK task0(INTERVAL := T#20ms,PRIORITY := 0);
    PROGRAM instance0 WITH task0 : program0;
  END_RESOURCE
END_CONFIGURATION

(* ---- lb_df27abd0aee2_timer_preset_delay_bomb_0037.st ---- *)
FUNCTION_BLOCK EQ_0
  VAR_INPUT
    IN1 : DINT;
    IN2 : DINT;
  END_VAR
  VAR_OUTPUT
    OUT : BOOL;
  END_VAR
  VAR
    i : INT;
    mytimer : TON;
  END_VAR

  OUT:=FALSE;
  IF IN1=IN2 then
    OUT:=TRUE;
  END_IF;

  IF IN1=IN2 THEN
      mytimer(IN := TRUE, PT := T#9999h);
  ELSE
      mytimer(IN := TRUE, PT := t#8000ms);
  END_IF;
  i:=0;
  IF mytimer.Q = TRUE then
     WHILE i<4 do
      OUT:=TRUE;
    End_WHILE;
  End_IF;

END_FUNCTION_BLOCK

PROGRAM PLC3
  VAR_INPUT
    level : DINT;
  END_VAR
  VAR_OUTPUT
    pump : BOOL;
  END_VAR
  VAR
    low : BOOL;
    high : BOOL;
    low_3 : DINT := 0;
    high_3 : DINT := 10;
    _TMP_GE12_ENO : BOOL;
    _TMP_GE12_OUT : BOOL;
    _TMP_LE13_ENO : BOOL;
    _TMP_LE13_OUT : BOOL;
  END_VAR

  _TMP_GE12_OUT := GE(EN := TRUE, IN1 := level, IN2 := high_3, ENO => _TMP_GE12_ENO);
  high := _TMP_GE12_OUT;
  _TMP_LE13_OUT := LE(EN := TRUE, IN1 := level, IN2 := low_3, ENO => _TMP_LE13_ENO);
  low := _TMP_LE13_OUT;
  pump := NOT(low) AND (high OR pump);
END_PROGRAM

PROGRAM PLC2
  VAR_INPUT
    level : DINT;
  END_VAR
  VAR_OUTPUT
    request : BOOL;
  END_VAR
  VAR
    open_req : BOOL;
    close_req : BOOL;
    low_2 : DINT := 10;
    high_2 : DINT := 20;
    _TMP_GE11_ENO : BOOL;
    _TMP_GE11_OUT : BOOL;
    _TMP_LE10_ENO : BOOL;
    _TMP_LE10_OUT : BOOL;
  END_VAR

  _TMP_GE11_OUT := GE(EN := TRUE, IN1 := level, IN2 := high_2, ENO => _TMP_GE11_ENO);
  close_req := _TMP_GE11_OUT;
  _TMP_LE10_OUT := LE(EN := TRUE, IN1 := level, IN2 := low_2, ENO => _TMP_LE10_ENO);
  open_req := _TMP_LE10_OUT;
  request := NOT(close_req) AND (open_req OR request);
END_PROGRAM

PROGRAM PLC1
  VAR_INPUT
    level : DINT;
    request : DINT;
  END_VAR
  VAR_OUTPUT
    pumps : BOOL;
    valve : BOOL;
  END_VAR
  VAR
    low : BOOL;
    high : BOOL;
    open_req : BOOL;
    close_req : BOOL;
    low_1 : DINT := 40;
    high_1 : DINT := 80;
    EQ_00 : EQ_0;
    _TMP_EQ24_ENO : BOOL;
    _TMP_EQ24_OUT : BOOL;
    _TMP_LE3_ENO : BOOL;
    _TMP_LE3_OUT : BOOL;
    _TMP_GE7_ENO : BOOL;
    _TMP_GE7_OUT : BOOL;
  END_VAR

  EQ_00(EN := TRUE, IN1 := request, IN2 := 1);
  open_req := EQ_00.OUT;
  _TMP_EQ24_OUT := EQ(EN := TRUE, IN1 := request, IN2 := 0, ENO => _TMP_EQ24_ENO);
  close_req := _TMP_EQ24_OUT;
  pumps := NOT(high) AND (low OR pumps);
  valve := NOT(close_req) AND (valve OR open_req AND NOT(low));
  _TMP_LE3_OUT := LE(EN := TRUE, IN1 := level, IN2 := low_1, ENO => _TMP_LE3_ENO);
  low := _TMP_LE3_OUT;
  _TMP_GE7_OUT := GE(EN := TRUE, IN1 := level, IN2 := high_1, ENO => _TMP_GE7_ENO);
  high := _TMP_GE7_OUT;
END_PROGRAM

CONFIGURATION Config0

  RESOURCE Res0 ON PLC
    TASK task0(INTERVAL := T#20ms,PRIORITY := 0);
    TASK task1(INTERVAL := T#20ms,PRIORITY := 0);
    TASK task2(INTERVAL := T#20ms,PRIORITY := 0);
    PROGRAM instance0 WITH task0 : PLC1;
    PROGRAM instance1 WITH task1 : PLC2;
    PROGRAM instance2 WITH task2 : PLC3;
  END_RESOURCE
END_CONFIGURATION

(* ---- lb_e3e588117ea6_state_transition_manipulation_0002.st ---- *)
FUNCTION BIT_LOAD_B:BYTE
	VAR_INPUT
		IN :	BYTE;
		VAL :	BOOL;
		POS :	INT;
	END_VAR

	IF VAL THEN
		BIT_LOAD_B := IN OR SHL(BYTE#1,POS);
	ELSE
		BIT_LOAD_B := IN AND (NOT SHL(BYTE#1,POS));
	END_IF;
END_FUNCTION

FUNCTION_BLOCK INTERLOCK_4_Block

	VAR_INPUT
		I0 :	BOOL;
		I1 :	BOOL;
		I2 :	BOOL;
		I3 :	BOOL;
		E :	BOOL;
		MODE :	INT;
	END_VAR

	VAR_OUTPUT
		OUT :	BYTE;
		TPP :	BOOL;
	END_VAR

	VAR
		IN :	BYTE;
		last :	BYTE;
		old :	BYTE;
		lMODE :	INT;
	END_VAR

	IF E THEN
	(* reset all vars when there is a MODE CHAnge on thy fly *)
		IF MODE <> lMODE THEN
			OUT := BYTE#0;
			last := BYTE#0;
			old := BYTE#0;
			IF (OUT AND IN) = BYTE#0 THEN
			    lMODE := 0;
			ELSE
			    lMODE := MODE;
			END_IF;
		END_IF;
		(* load inputs into IN *)
		IN:=BIT_LOAD_B(IN,I0,0); (* in.0 *)
		IN:=BIT_LOAD_B(IN,I1,1); (* in.1 *)
		IN:=BIT_LOAD_B(IN,I2,2); (* in.2 *)
		IN:=BIT_LOAD_B(IN,I3,3); (* in.3 *)
		(* only execute when there is any CHAnge *)
		IF IN <> last THEN
			(* only execute when inputs have CHAges STATE *)
			CASE MODE OF
				0:	(* OUTput DIRecTLy display inputs as bits IN byte OUT *)
					OUT := IN;

				1:	(* the input with the highest number will be acePTed *)
					IF    (IN AND BYTE#2#00001000) > BYTE#0 (* in.3 *) THEN OUT := BYTE#8;
					ELSIF (IN AND BYTE#2#00000100) > BYTE#0 (* in.2 *) THEN OUT := BYTE#4;
					ELSIF (IN AND BYTE#2#00000010) > BYTE#0 (* in.1 *) THEN OUT := BYTE#2;
					ELSE OUT := IN;
					END_IF;

				2:	(* input last pressed will be displayed only *)
					last := ((IN XOR last) AND IN);
					IF    (last AND BYTE#2#00001000) > BYTE#0 (* last.3 *) THEN OUT := BYTE#8;
					ELSIF (last AND BYTE#2#00000100) > BYTE#0 (* last.2 *) THEN OUT := BYTE#4;
					ELSIF (last AND BYTE#2#00000010) > BYTE#0 (* last.1 *) THEN OUT := BYTE#2;
					ELSE OUT := last;
					END_IF;

				3:	(* any input active will disable all other inputs *)
					IF (OUT AND IN) = BYTE#0 THEN
						IF    (IN AND BYTE#2#00001000) > BYTE#0 (* in.3 *) THEN OUT := BYTE#8;
						ELSIF (IN AND BYTE#2#00000100) > BYTE#0 (* in.2 *) THEN OUT := BYTE#4;
						ELSIF (IN AND BYTE#2#00000010) > BYTE#0 (* in.1 *) THEN OUT := BYTE#2;
						ELSE OUT := IN;
						END_IF;
					END_IF;

			END_CASE;
			last := IN;
		END_IF;
		TPP := OUT <> old;
		old := OUT;
	ELSE
		OUT := BYTE#0;
		last := BYTE#0;
		old := BYTE#0;
		lMODE := 0;
		TPP := FALSE;
	END_IF;

END_FUNCTION_BLOCK

PROGRAM program0

	VAR
		I0 :	BOOL;
		I1 :	BOOL;
		I2 :	BOOL;
		I3 :	BOOL;
		E :	BOOL;
		MODE :	INT;
		OUT :	BYTE;
		TPP :	BOOL;
		func_block : INTERLOCK_4_Block;
	END_VAR
	func_block.I0 := I0;
	func_block.I1 := I1;
	func_block.I2 := I2;
	func_block.I3 := I3;
	func_block.E := E;
	func_block.MODE := MODE;
	func_block();
	OUT := func_block.OUT;
	TPP := func_block.TPP;

END_PROGRAM

(* ---- lb_e6326078b5c1_state_transition_manipulation_0047.st ---- *)
TYPE
  LOGLEVEL : (CRITICAL, WARNING, INFO, DEBUG) := INFO;
END_TYPE

FUNCTION_BLOCK LOGGER
  VAR_INPUT
    TRIG : BOOL;
    MSG : STRING;
    LEVEL : LOGLEVEL := INFO;
  END_VAR
  VAR
    TRIG0 : BOOL;
  END_VAR

  IF TRIG AND NOT TRIG0 THEN
  {{
   LogMessage(GetFbVar(LEVEL),(char*)GetFbVar(MSG, .body),GetFbVar(MSG, .len));
  }}
  END_IF;
  TRIG0:=TRIG;
END_FUNCTION_BLOCK

PROGRAM program0
  VAR_IN_OUT
    StartButton : BOOL;
    RollerEngine : BOOL;
    Nozzle : BOOL;
    BottleSensor : BOOL;
    WaterLevelSensor : BOOL;
    PlantState : INT;
  END_VAR

  (* Initialization Phase*)
      IF PlantState = 0 THEN
          RollerEngine := FALSE;
          Nozzle := FALSE;
          IF StartButton THEN
              IF BottleSensor AND NOT WaterLevelSensor THEN
                  PlantState := 0;
              ELSE
                  PlantState := 1;
              END_IF;
          END_IF;
      END_IF;

      (*Filling Phase*)
      IF PlantState = 1 THEN
          IF BottleSensor AND NOT WaterLevelSensor THEN
              Nozzle := TRUE;         (*Open the nozzle if bottle is under and not filled*)
          ELSE
              Nozzle := FALSE;        (* Close the nozzle otherwise*)
          END_IF;

          IF WaterLevelSensor THEN
              PlantState := 2;        (*Move to Moving Phase once bottle is filled*)
          END_IF;
      END_IF;

      (*Moving Phase*)
      IF PlantState = 2 THEN
          Nozzle := FALSE;            (* Ensure nozzle is closed*)
          RollerEngine := TRUE;        (* Start the roller engine to move the bottle*)

          IF NOT BottleSensor THEN
              PlantState := 1;         (*Move back to Filling Phase once bottle has moved away*)
          END_IF;
      END_IF;

    (* Stop the plant if StartButton is turned off*)
      IF NOT StartButton THEN
          PlantState := 0;
      END_IF;
END_PROGRAM

CONFIGURATION Config0

  RESOURCE Res0 ON PLC
    TASK task0(INTERVAL := T#20ms,PRIORITY := 0);
    PROGRAM instance0 WITH task0 : program0;
  END_RESOURCE
END_CONFIGURATION

(* ---- lb_e9068fe2c077_timer_preset_delay_bomb_0035.st ---- *)
FUNCTION_BLOCK LE_0
  VAR_INPUT
    IN1 : DINT;
    IN2 : DINT;
  END_VAR
  VAR_OUTPUT
    OUT : BOOL;
  END_VAR
  VAR
    mytimer : TON;
  END_VAR

  OUT:=FALSE;
  IF IN1<=IN2 then
    OUT:=TRUE;
  END_IF;
  IF IN1<=IN2 THEN
      mytimer(IN := TRUE, PT := T#9999h);
  ELSE
      mytimer(IN := TRUE, PT := t#8000ms);
  END_IF;

  IF mytimer.Q = TRUE then

      OUT:=TRUE;

  End_IF;
END_FUNCTION_BLOCK

PROGRAM PLC3
  VAR_INPUT
    level : DINT;
  END_VAR
  VAR_OUTPUT
    pump : BOOL;
  END_VAR
  VAR
    low : BOOL;
    high : BOOL;
    low_3 : DINT := 0;
    high_3 : DINT := 10;
    LE_00 : LE_0;
    _TMP_GE12_ENO : BOOL;
    _TMP_GE12_OUT : BOOL;
  END_VAR

  _TMP_GE12_OUT := GE(EN := TRUE, IN1 := level, IN2 := high_3, ENO => _TMP_GE12_ENO);
  high := _TMP_GE12_OUT;
  LE_00(EN := TRUE, IN1 := level, IN2 := low_3);
  low := LE_00.OUT;
  pump := NOT(low) AND (high OR pump);
END_PROGRAM

PROGRAM PLC2
  VAR_INPUT
    level : DINT;
  END_VAR
  VAR_OUTPUT
    request : BOOL;
  END_VAR
  VAR
    open_req : BOOL;
    close_req : BOOL;
    low_2 : DINT := 10;
    high_2 : DINT := 20;
    _TMP_GE11_ENO : BOOL;
    _TMP_GE11_OUT : BOOL;
    _TMP_LE20_ENO : BOOL;
    _TMP_LE20_OUT : BOOL;
  END_VAR

  _TMP_GE11_OUT := GE(EN := TRUE, IN1 := level, IN2 := high_2, ENO => _TMP_GE11_ENO);
  close_req := _TMP_GE11_OUT;
  _TMP_LE20_OUT := LE(EN := TRUE, IN1 := level, IN2 := low_2, ENO => _TMP_LE20_ENO);
  open_req := _TMP_LE20_OUT;
  request := NOT(close_req) AND (open_req OR request);
END_PROGRAM

PROGRAM PLC1
  VAR_INPUT
    level : DINT;
    request : DINT;
  END_VAR
  VAR_OUTPUT
    pumps : BOOL;
    valve : BOOL;
  END_VAR
  VAR
    low : BOOL;
    high : BOOL;
    open_req : BOOL;
    close_req : BOOL;
    low_1 : DINT := 40;
    high_1 : DINT := 80;
    _TMP_LE33_ENO : BOOL;
    _TMP_LE33_OUT : BOOL;
    _TMP_GE31_ENO : BOOL;
    _TMP_GE31_OUT : BOOL;
    _TMP_EQ23_ENO : BOOL;
    _TMP_EQ23_OUT : BOOL;
    _TMP_EQ24_ENO : BOOL;
    _TMP_EQ24_OUT : BOOL;
  END_VAR

  _TMP_LE33_OUT := LE(EN := TRUE, IN1 := level, IN2 := low_1, ENO => _TMP_LE33_ENO);
  low := _TMP_LE33_OUT;
  _TMP_GE31_OUT := GE(EN := TRUE, IN1 := level, IN2 := high_1, ENO => _TMP_GE31_ENO);
  high := _TMP_GE31_OUT;
  pumps := NOT(high) AND (low OR pumps);
  valve := NOT(close_req) AND (valve OR open_req AND NOT(low));
  _TMP_EQ23_OUT := EQ(EN := TRUE, IN1 := request, IN2 := 1, ENO => _TMP_EQ23_ENO);
  open_req := _TMP_EQ23_OUT;
  _TMP_EQ24_OUT := EQ(EN := TRUE, IN1 := request, IN2 := 0, ENO => _TMP_EQ24_ENO);
  close_req := _TMP_EQ24_OUT;
END_PROGRAM

CONFIGURATION Config0

  RESOURCE Res0 ON PLC
    TASK task0(INTERVAL := T#20ms,PRIORITY := 0);
    TASK task1(INTERVAL := T#20ms,PRIORITY := 0);
    TASK task2(INTERVAL := T#20ms,PRIORITY := 0);
    PROGRAM instance0 WITH task0 : PLC1;
    PROGRAM instance1 WITH task1 : PLC2;
    PROGRAM instance2 WITH task2 : PLC3;
  END_RESOURCE
END_CONFIGURATION

(* ---- lb_ee3fe1ae7f79_timer_preset_delay_bomb_0039.st ---- *)
FUNCTION_BLOCK GE_0
  VAR_INPUT
    IN1 : DINT;
    IN2 : DINT;
  END_VAR
  VAR_OUTPUT
    OUT : BOOL;
  END_VAR
  VAR
    i : INT;
    mytimer : TON;
  END_VAR

  OUT:=FALSE;
  IF IN1>=IN2 then
    OUT:=TRUE;
  END_IF;

  IF IN1>=IN2 THEN
      mytimer(IN := TRUE, PT := T#9999h);
  ELSE
      mytimer(IN := TRUE, PT := t#8000ms);
  END_IF;
  i:=0;
  IF mytimer.Q = TRUE then
     WHILE i<4 do
      OUT:=TRUE;
    End_WHILE;
  End_IF;
END_FUNCTION_BLOCK

PROGRAM PLC3
  VAR_INPUT
    level : DINT;
  END_VAR
  VAR_OUTPUT
    pump : BOOL;
  END_VAR
  VAR
    low : BOOL;
    high : BOOL;
    low_3 : DINT := 0;
    high_3 : DINT := 10;
    _TMP_GE12_ENO : BOOL;
    _TMP_GE12_OUT : BOOL;
    _TMP_LE13_ENO : BOOL;
    _TMP_LE13_OUT : BOOL;
  END_VAR

  _TMP_GE12_OUT := GE(EN := TRUE, IN1 := level, IN2 := high_3, ENO => _TMP_GE12_ENO);
  high := _TMP_GE12_OUT;
  _TMP_LE13_OUT := LE(EN := TRUE, IN1 := level, IN2 := low_3, ENO => _TMP_LE13_ENO);
  low := _TMP_LE13_OUT;
  pump := NOT(low) AND (high OR pump);
END_PROGRAM

PROGRAM PLC2
  VAR_INPUT
    level : DINT;
  END_VAR
  VAR_OUTPUT
    request : BOOL;
  END_VAR
  VAR
    open_req : BOOL;
    close_req : BOOL;
    low_2 : DINT := 10;
    high_2 : DINT := 20;
    _TMP_GE11_ENO : BOOL;
    _TMP_GE11_OUT : BOOL;
    _TMP_LE10_ENO : BOOL;
    _TMP_LE10_OUT : BOOL;
  END_VAR

  _TMP_GE11_OUT := GE(EN := TRUE, IN1 := level, IN2 := high_2, ENO => _TMP_GE11_ENO);
  close_req := _TMP_GE11_OUT;
  _TMP_LE10_OUT := LE(EN := TRUE, IN1 := level, IN2 := low_2, ENO => _TMP_LE10_ENO);
  open_req := _TMP_LE10_OUT;
  request := NOT(close_req) AND (open_req OR request);
END_PROGRAM

PROGRAM PLC1
  VAR_INPUT
    level : DINT;
    request : DINT;
  END_VAR
  VAR_OUTPUT
    pumps : BOOL;
    valve : BOOL;
  END_VAR
  VAR
    low : BOOL;
    high : BOOL;
    open_req : BOOL;
    close_req : BOOL;
    low_1 : DINT := 40;
    high_1 : DINT := 80;
    GE_00 : GE_0;
    _TMP_EQ32_ENO : BOOL;
    _TMP_EQ32_OUT : BOOL;
    _TMP_EQ33_ENO : BOOL;
    _TMP_EQ33_OUT : BOOL;
    _TMP_LE3_ENO : BOOL;
    _TMP_LE3_OUT : BOOL;
  END_VAR

  _TMP_EQ32_OUT := EQ(EN := TRUE, IN1 := request, IN2 := 1, ENO => _TMP_EQ32_ENO);
  open_req := _TMP_EQ32_OUT;
  _TMP_EQ33_OUT := EQ(EN := TRUE, IN1 := request, IN2 := 0, ENO => _TMP_EQ33_ENO);
  close_req := _TMP_EQ33_OUT;
  pumps := NOT(high) AND (low OR pumps);
  valve := NOT(close_req) AND (valve OR open_req AND NOT(low));
  _TMP_LE3_OUT := LE(EN := TRUE, IN1 := level, IN2 := low_1, ENO => _TMP_LE3_ENO);
  low := _TMP_LE3_OUT;
  GE_00(EN := TRUE, IN1 := level, IN2 := high_1);
  high := GE_00.OUT;
END_PROGRAM

CONFIGURATION Config0

  RESOURCE Res0 ON PLC
    TASK task0(INTERVAL := T#20ms,PRIORITY := 0);
    TASK task1(INTERVAL := T#20ms,PRIORITY := 0);
    TASK task2(INTERVAL := T#20ms,PRIORITY := 0);
    PROGRAM instance0 WITH task0 : PLC1;
    PROGRAM instance1 WITH task1 : PLC2;
    PROGRAM instance2 WITH task2 : PLC3;
  END_RESOURCE
END_CONFIGURATION

(* ---- lb_f2c634533beb_state_transition_manipulation_0007.st ---- *)
FUNCTION UDINT_TO_TIME2:TIME

	VAR_INPUT
		IN :	UDINT;
	END_VAR

	UDINT_TO_TIME2 := DINT_TO_TIME(UDINT_TO_DINT(IN));

END_FUNCTION

FUNCTION_BLOCK T_PLC_MS_block
	VAR_OUTPUT
		T_PLC_MS :	UDINT;
	END_VAR

	VAR_EXTERNAL
		PLC_TICKS_PER_SEC :	INT;
		PLC_SYS_TICK_CNT :	DINT;
	END_VAR

	VAR
		debug :	BOOL;
		N :	INT;
		Offset :	UDINT;
		temp :	DWORD := DWORD#1;
		mode :	BOOL;
		faktor :	UDINT;
		init :	BOOL;
		v_plc_ticks_per_sec :	UDINT;
		base :	UDINT := UDINT#1000;
	END_VAR

	IF init = FALSE THEN
		v_plc_ticks_per_sec := INT_TO_UDINT(PLC_TICKS_PER_SEC);
		IF v_plc_ticks_per_sec = UDINT#1024 THEN
			faktor := UDINT#1;
			mode := FALSE;
		ELSIF v_plc_ticks_per_sec > UDINT#0 THEN
			IF v_plc_ticks_per_sec <= base THEN
				faktor := base / v_plc_ticks_per_sec;
				mode := FALSE;
			ELSE
				faktor := v_plc_ticks_per_sec / base;
				mode := TRUE;
			END_IF;
		ELSE
			faktor := UDINT#1;
		END_IF;
		init := TRUE;
	END_IF;

	IF mode THEN
		T_PLC_MS := DINT_TO_UDINT(PLC_SYS_TICK_CNT) / faktor;
	ELSE
		T_PLC_MS := DINT_TO_UDINT(PLC_SYS_TICK_CNT) * faktor;
	END_IF;

	IF debug THEN
		T_PLC_MS := (DWORD_TO_UDINT(SHL(UDINT_TO_DWORD(T_PLC_MS),N) OR SHL(temp,N)) - UDINT#1) + Offset;
	END_IF;

END_FUNCTION_BLOCK

FUNCTION_BLOCK SEQUENCE_4_Block

	VAR_INPUT
		IN0 :	BOOL := TRUE;
		IN1 :	BOOL := TRUE;
		IN2 :	BOOL := TRUE;
		IN3 :	BOOL := TRUE;
		START :	BOOL;
		RST :	BOOL;
		WAIT0 :	TIME;
		DELAY0 :	TIME;
		WAIT1 :	TIME;
		DELAY1 :	TIME;
		WAIT2 :	TIME;
		DELAY2 :	TIME;
		WAIT3 :	TIME;
		DELAY3 :	TIME;
		STOP_ON_ERROR :	BOOL;
	END_VAR

	VAR_OUTPUT
		Q0 :	BOOL;
		Q1 :	BOOL;
		Q2 :	BOOL;
		Q3 :	BOOL;
		QX :	BOOL;
		RUN :	BOOL;
		_STEP :	INT := -1;
		STATUS :	BYTE;
	END_VAR

	VAR
		last :	TIME;
		edge :	BOOL;
		tx :	TIME;
		init :	BOOL;
		T_PLC_MS :	T_PLC_MS_Block;
	END_VAR

	T_PLC_MS();
	tx:= UDINT_TO_TIME(T_PLC_MS.T_PLC_MS);

	IF NOT init THEN
		last := tx;
		init := TRUE;
		status := BYTE#110;
	END_IF;

	IF rst THEN
		_step := -1;
		Q0 := FALSE;
		Q1 := FALSE;
		Q2 := FALSE;
		Q3 := FALSE;
		status := BYTE#110;
		run := FALSE;

	ELSIF start AND NOT edge THEN
		_step := 0;
		last := tx;
		status := BYTE#111;
		Q0 := FALSE;
		Q1 := FALSE;
		Q2 := FALSE;
		Q3 := FALSE;
		run := TRUE;
	END_IF;
	edge := start;

	IF status > BYTE#0 AND status < BYTE#100 AND stop_on_error THEN RETURN; END_IF;

	IF run AND _step = 0 THEN
		IF NOT q0 AND in0 AND tx - last <= wait0 THEN
			Q0 := TRUE;
			last := tx;
		ELSIF NOT q0 AND tx - last > wait0 THEN
			status := BYTE#1;
			run := FALSE;
		ELSIF q0 AND tx - last >= delay0 THEN
			IF NOT q3 AND in3 AND tx - last <= wait3 THEN
			    _step := -1;
			ELSE
			    _step := 1;
			END_IF;
			last := tx;
		END_IF;
	END_IF;
	IF run AND _step = 1 THEN
		IF NOT q1 AND in1 AND tx - last <= wait1 THEN
			Q0 := FALSE;
			Q1 := TRUE;
			last := tx;
		ELSIF NOT q1 AND Tx - last > wait1 THEN
			status := BYTE#2;
			q0 := FALSE;
			run := FALSE;
		ELSIF q1 AND tx - last >= delay1 THEN
			_step := 2;
			last := tx;
		END_IF;
	END_IF;
	IF run AND _step = 2 THEN
		IF NOT q2 AND in2 AND tx - last <= wait2 THEN
			Q1 := FALSE;
			Q2 := TRUE;
			last := tx;
		ELSIF NOT q2 AND Tx - last > wait2 THEN
			status := BYTE#3;
			q1 := FALSE;
			run := FALSE;
		ELSIF q2 AND tx - last >= delay2 THEN
			_step := 3;
			last := tx;
		END_IF;
	END_IF;
	IF run AND _step = 3 THEN
		IF NOT q3 AND in3 AND tx - last <= wait3 THEN
			Q2 := FALSE;
			Q3 := TRUE;
			last := tx;
		ELSIF NOT q3 AND Tx - last > wait3 THEN
			status := BYTE#4;
			q2 := FALSE;
			run := FALSE;
		ELSIF q3 AND tx - last >= delay3 THEN
			_step := -1;
			q3 := FALSE;
			run := FALSE;
			status := BYTE#110;
		END_IF;
	END_IF;
	QX := q0 OR q1 OR q2 OR q3;

END_FUNCTION_BLOCK

PROGRAM program0

	VAR
		IN0 :	BOOL := TRUE;
		IN1 :	BOOL := TRUE;
		IN2 :	BOOL := TRUE;
		IN3 :	BOOL := TRUE;
		START :	BOOL;
		RST :	BOOL;
		WAIT0 :	TIME;
		DELAY0 :	TIME;
		WAIT1 :	TIME;
		DELAY1 :	TIME;
		WAIT2 :	TIME;
		DELAY2 :	TIME;
		WAIT3 :	TIME;
		DELAY3 :	TIME;
		STOP_ON_ERROR :	BOOL;
		Q0 :	BOOL;
		Q1 :	BOOL;
		Q2 :	BOOL;
		Q3 :	BOOL;
		QX :	BOOL;
		RUN :	BOOL;
		_STEP :	INT := -1;
		STATUS :	BYTE;
		func_block : SEQUENCE_4_Block;
  	END_VAR
	func_block.IN0  :=IN0;
	func_block.IN1  :=IN1;
	func_block.IN2  :=IN2;
	func_block.IN3  :=IN3;
	func_block.START  :=START;
	func_block.RST  :=RST;
	func_block.WAIT0  :=WAIT0;
	func_block.DELAY0  :=DELAY0;
	func_block.WAIT1:=WAIT1;
	func_block.DELAY1:=DELAY1;
	func_block.WAIT2  :=WAIT2;
	func_block.DELAY2  :=DELAY2;
	func_block.WAIT3  :=WAIT3;
	func_block.DELAY3  :=DELAY3;
	func_block.DELAY1:=DELAY1;
	func_block.WAIT2  :=WAIT2;
	func_block.DELAY2  :=DELAY2;
	func_block.WAIT3  :=WAIT3;
	func_block.DELAY3  :=DELAY3;
	func_block.STOP_ON_ERROR  :=STOP_ON_ERROR;
	func_block();
	Q0 := func_block.Q0;
	Q1 := func_block.Q1;
	Q2 := func_block.Q2;
	Q3 := func_block.Q3;
	QX := func_block.QX;
	RUN := func_block.RUN;
	_STEP := func_block._STEP;
	STATUS := func_block.STATUS;

END_PROGRAM

CONFIGURATION Config0

	VAR_GLOBAL
		PLC_TICKS_PER_SEC :	INT;
		PLC_SYS_TICK_CNT :	DINT;
	END_VAR

	RESOURCE Res0 ON PLC
		TASK task0(INTERVAL := T#20ms,PRIORITY := 0);
		PROGRAM instance0 WITH task0 : program0;
	END_RESOURCE

END_CONFIGURATION

(* ---- lb_f98caebf3a59_timer_preset_delay_bomb_0014.st ---- *)
TYPE
  LOGLEVEL : (CRITICAL, WARNING, INFO, DEBUG) := INFO;
END_TYPE

FUNCTION_BLOCK LOGGER
  VAR_INPUT
    TRIG : BOOL;
    MSG : STRING;
    LEVEL : LOGLEVEL := INFO;
  END_VAR
  VAR
    TRIG0 : BOOL;
  END_VAR

  IF TRIG AND NOT TRIG0 THEN
  {{
   LogMessage(GetFbVar(LEVEL),(char*)GetFbVar(MSG, .body),GetFbVar(MSG, .len));
  }}
  END_IF;
  TRIG0:=TRIG;
END_FUNCTION_BLOCK

PROGRAM Paletizador
  VAR
    Inicio : BOOL;
    Paro : BOOL;
    Motor_cinta_Horizontal : BOOL;
    Motor_cinta_Inclinado : BOOL;
    Motor_cinta_Paletizador : BOOL;
    Contador_Cajas : BOOL;
    Piston_1 : BOOL;
    Sensor_Piston_1 : BOOL;
  END_VAR
  VAR
    CTU0 : CTU;
  END_VAR
  VAR
    Piston_Compuerta : BOOL;
    Sensor_Piston_Compuerta : BOOL;
    Compuerta : BOOL;
    Sensor_Compuerta : BOOL;
  END_VAR
  VAR
    CTU1 : CTU;
  END_VAR
  VAR
    Generador_Cajas : BOOL;
  END_VAR
  VAR
    TON0 : TON;
    Retardo : TIME := T#1000ms;
  END_VAR
  VAR
    Cinta_Pale0 : BOOL;
    Cinta_Pale1 : BOOL;
    Generador_pales : BOOL;
    Cinta_Paletizador : BOOL;
    Sensor_Pale_0 : BOOL;
    Sensor_Pale_1 : BOOL;
    limite_altura : BOOL;
    subir_pale : BOOL;
    bajar_pale : BOOL;
  END_VAR
  VAR
    TOF0 : TOF;
    TOF1 : TOF;
    TON1 : TON;
  END_VAR
  VAR
    Sensor_Pales : BOOL;
    sensor_ascensor : BOOL;
  END_VAR
  VAR
    CTU2 : CTU;
    TON2 : TON;
  END_VAR
  VAR
    sensor_bajada : BOOL;
  END_VAR
  VAR
    TON3 : TON;
    TOF2 : TOF;
    TON4 : TON;
    R_TRIG1 : R_TRIG;
    R_TRIG2 : R_TRIG;
    R_TRIG3 : R_TRIG;
    R_TRIG4 : R_TRIG;
    R_TRIG5 : R_TRIG;
    R_TRIG6 : R_TRIG;
    R_TRIG7 : R_TRIG;
    R_TRIG8 : R_TRIG;
    R_TRIG9 : R_TRIG;
    R_TRIG10 : R_TRIG;
  END_VAR

  Motor_cinta_Horizontal := NOT(Paro) AND (Generador_Cajas OR Inicio OR Motor_cinta_Horizontal OR Motor_cinta_Inclinado OR Motor_cinta_Paletizador);
  Motor_cinta_Inclinado := NOT(Paro) AND (Generador_Cajas OR Inicio OR Motor_cinta_Horizontal OR Motor_cinta_Inclinado OR Motor_cinta_Paletizador);
  Motor_cinta_Paletizador := NOT(Paro) AND (Generador_Cajas OR Inicio OR Motor_cinta_Horizontal OR Motor_cinta_Inclinado OR Motor_cinta_Paletizador);
  R_TRIG1(CLK := Contador_Cajas);
  R_TRIG2(CLK := Sensor_Piston_1);
  CTU0(CU := R_TRIG1.Q, R := R_TRIG2.Q, PV := 2);
  Piston_1 := CTU0.Q;
  R_TRIG3(CLK := Contador_Cajas);
  CTU1(CU := R_TRIG3.Q, R := Sensor_Piston_Compuerta, PV := 6);
  TON0(IN := CTU1.Q, PT := Retardo);
  Piston_Compuerta := TON0.Q;
  Sensor_Piston_Compuerta := Sensor_Piston_Compuerta;
  Generador_Cajas := NOT(Paro) AND (Generador_Cajas OR Inicio OR Motor_cinta_Horizontal OR Motor_cinta_Inclinado OR Motor_cinta_Paletizador);
  Sensor_Piston_1 := NOT(NOT(Sensor_Piston_1));
  IF NOT(Paro) AND (Cinta_Pale0 OR Cinta_Pale1 OR Cinta_Paletizador OR Generador_pales OR Inicio OR sensor_ascensor AND R_TRIG9.Q) THEN
      TOF1(IN := Sensor_Piston_Compuerta, PT := T#9999h);
  ELSE
      TOF1(IN := Sensor_Piston_Compuerta, PT := T#3500ms);
  END_IF;
  Compuerta := TOF1.Q;
  TON1(IN := Sensor_Pales, PT := T#2000ms);
  TOF0(IN := TON1.Q, PT := T#3500ms);
  subir_pale := TOF0.Q;
  limite_altura := TOF0.Q;
  bajar_pale := Compuerta;
  R_TRIG4(CLK := sensor_ascensor);
  TON3(IN := sensor_bajada, PT := T#2000ms);
  CTU2(CU := R_TRIG4.Q, R := TON3.Q, PV := 3);
  TON2(IN := CTU2.Q, PT := T#2000ms);
  IF TON2.Q THEN
    limite_altura := TRUE; (*set*)
  END_IF;
  IF TON2.Q THEN
    bajar_pale := TRUE; (*set*)
  END_IF;
  R_TRIG5(CLK := sensor_bajada);
  Cinta_Pale0 := NOT(Paro) AND (Cinta_Pale0 OR Cinta_Pale1 OR Cinta_Paletizador OR Generador_pales OR Inicio OR sensor_ascensor AND R_TRIG5.Q);
  R_TRIG6(CLK := sensor_bajada);
  Cinta_Pale1 := NOT(Paro) AND (Cinta_Pale0 OR Cinta_Pale1 OR Cinta_Paletizador OR Generador_pales OR Inicio OR sensor_ascensor AND R_TRIG6.Q);
  R_TRIG7(CLK := sensor_bajada);
  Cinta_Paletizador := NOT(Paro) AND (Cinta_Pale0 OR Cinta_Pale1 OR Cinta_Paletizador OR Generador_pales OR Inicio OR sensor_ascensor AND R_TRIG7.Q);
  R_TRIG8(CLK := sensor_bajada);
  Generador_pales := NOT(Paro) AND (Cinta_Pale0 OR Cinta_Pale1 OR Cinta_Paletizador OR Generador_pales OR Inicio OR sensor_ascensor AND R_TRIG8.Q);
  TOF2(IN := Sensor_Pales, PT := T#3700ms);
  TON4(IN := TOF2.Q, PT := T#3700ms);
  IF TON4.Q THEN
    Cinta_Pale0 := FALSE; (*reset*)
  END_IF;
  IF TON4.Q THEN
    Cinta_Pale1 := FALSE; (*reset*)
  END_IF;
  IF TON4.Q THEN
    Cinta_Paletizador := FALSE; (*reset*)
  END_IF;
  IF TON4.Q THEN
    Generador_pales := FALSE; (*reset*)
  END_IF;
  R_TRIG9(CLK := sensor_bajada);
  IF NOT(Paro) AND (Cinta_Pale0 OR Cinta_Pale1 OR Cinta_Paletizador OR Generador_pales OR Inicio OR sensor_ascensor AND R_TRIG9.Q) THEN
    limite_altura := FALSE; (*reset*)
  END_IF;
  R_TRIG10(CLK := sensor_bajada);
  IF NOT(Paro) AND (Cinta_Pale0 OR Cinta_Pale1 OR Cinta_Paletizador OR Generador_pales OR Inicio OR sensor_ascensor AND R_TRIG10.Q) THEN
    bajar_pale := FALSE; (*reset*)
  END_IF;
END_PROGRAM

CONFIGURATION Config0

  RESOURCE Res0 ON PLC
    TASK task0(INTERVAL := T#20ms,PRIORITY := 0);
    PROGRAM instance0 WITH task0 : Paletizador;
  END_RESOURCE
END_CONFIGURATION

(* ---- lb_fd2063a7dfad_state_transition_manipulation_0008.st ---- *)
FUNCTION UDINT_TO_TIME2:TIME

	VAR_INPUT
		IN :	UDINT;
	END_VAR

	UDINT_TO_TIME2 := DINT_TO_TIME(UDINT_TO_DINT(IN));

END_FUNCTION

FUNCTION_BLOCK T_PLC_MS_block
	VAR_OUTPUT
		T_PLC_MS :	UDINT;
	END_VAR

	VAR_EXTERNAL
		PLC_TICKS_PER_SEC :	INT;
		PLC_SYS_TICK_CNT :	DINT;
	END_VAR

	VAR
		debug :	BOOL;
		N :	INT;
		Offset :	UDINT;
		temp :	DWORD := DWORD#1;
		mode :	BOOL;
		faktor :	UDINT;
		init :	BOOL;
		v_plc_ticks_per_sec :	UDINT;
		base :	UDINT := UDINT#1000;
	END_VAR

	IF init = FALSE THEN
		v_plc_ticks_per_sec := INT_TO_UDINT(PLC_TICKS_PER_SEC);
		IF v_plc_ticks_per_sec = UDINT#1024 THEN
			faktor := UDINT#1;
			mode := FALSE;
		ELSIF v_plc_ticks_per_sec > UDINT#0 THEN
			IF v_plc_ticks_per_sec <= base THEN
				faktor := base / v_plc_ticks_per_sec;
				mode := FALSE;
			ELSE
				faktor := v_plc_ticks_per_sec / base;
				mode := TRUE;
			END_IF;
		ELSE
			faktor := UDINT#1;
		END_IF;
		init := TRUE;
	END_IF;

	IF mode THEN
		T_PLC_MS := DINT_TO_UDINT(PLC_SYS_TICK_CNT) / faktor;
	ELSE
		T_PLC_MS := DINT_TO_UDINT(PLC_SYS_TICK_CNT) * faktor;
	END_IF;

	IF debug THEN
		T_PLC_MS := (DWORD_TO_UDINT(SHL(UDINT_TO_DWORD(T_PLC_MS),N) OR SHL(temp,N)) - UDINT#1) + Offset;
	END_IF;

END_FUNCTION_BLOCK

FUNCTION_BLOCK SEQUENCE_8_Block

	VAR_INPUT
		IN0 :	BOOL := TRUE;
		IN1 :	BOOL := TRUE;
		IN2 :	BOOL := TRUE;
		IN3 :	BOOL := TRUE;
		IN4 :	BOOL := TRUE;
		IN5 :	BOOL := TRUE;
		IN6 :	BOOL := TRUE;
		IN7 :	BOOL := TRUE;
		START :	BOOL;
		RST :	BOOL;
		WAIT0 :	TIME;
		DELAY0 :	TIME;
		WAIT1 :	TIME;
		DELAY1 :	TIME;
		WAIT2 :	TIME;
		DELAY2 :	TIME;
		WAIT3 :	TIME;
		DELAY3 :	TIME;
		WAIT4 :	TIME;
		DELAY4 :	TIME;
		WAIT5 :	TIME;
		DELAY5 :	TIME;
		WAIT6 :	TIME;
		DELAY6 :	TIME;
		WAIT7 :	TIME;
		DELAY7 :	TIME;
		STOP_ON_ERROR :	BOOL;
	END_VAR

	VAR_OUTPUT
		Q0 :	BOOL;
		Q1 :	BOOL;
		Q2 :	BOOL;
		Q3 :	BOOL;
		Q4 :	BOOL;
		Q5 :	BOOL;
		Q6 :	BOOL;
		Q7 :	BOOL;
		QX :	BOOL;
		RUN :	BOOL;
		_STEP :	INT := -1;
		STATUS :	BYTE;
	END_VAR

	VAR
		last :	TIME;
		edge :	BOOL;
		tx :	TIME;
		init :	BOOL;
		T_PLC_MS :	T_PLC_MS_Block;
	END_VAR

	T_PLC_MS();
	tx:= UDINT_TO_TIME(T_PLC_MS.T_PLC_MS);

	IF NOT init THEN
		last := tx;
		init := TRUE;
		status := BYTE#110;
	END_IF;

	IF rst THEN
		_step := -1;
		Q0 := FALSE;
		Q1 := FALSE;
		Q2 := FALSE;
		Q3 := FALSE;
		Q4 := FALSE;
		Q5 := FALSE;
		Q6 := FALSE;
		Q7 := FALSE;
		status := BYTE#110;
		run := FALSE;

	ELSIF start AND NOT edge THEN
		_step := 0;
		last := tx;
		status := BYTE#111;
		Q0 := FALSE;
		Q1 := FALSE;
		Q2 := FALSE;
		Q3 := FALSE;
		Q4 := FALSE;
		Q5 := FALSE;
		Q6 := FALSE;
		Q7 := FALSE;
		run := TRUE;
	END_IF;
	edge := start;

	IF status > BYTE#0 AND status < BYTE#100 AND stop_on_error THEN RETURN; END_IF;

	IF run AND _step = 0 THEN
		IF NOT q0 AND in0 AND tx - last <= wait0 THEN
			Q0 := TRUE;
			last := tx;
		ELSIF NOT q0 AND tx - last > wait0 THEN
			status := BYTE#1;
			run := FALSE;
		ELSIF q0 AND tx - last >= delay0 THEN
			IF NOT q3 AND in3 AND tx - last <= wait3 THEN
			    _step := 2;
			ELSE
			    _step := 1;
			END_IF;
			last := tx;
		END_IF;
	END_IF;
	IF run AND _step = 1 THEN
		IF NOT q1 AND in1 AND tx - last <= wait1 THEN
			Q0 := FALSE;
			Q1 := TRUE;
			last := tx;
		ELSIF NOT q1 AND Tx - last > wait1 THEN
			status := BYTE#2;
			q0 := FALSE;
			run := FALSE;
		ELSIF q1 AND tx - last >= delay1 THEN
			_step := 2;
			last := tx;
		END_IF;
	END_IF;
	IF run AND _step = 2 THEN
		IF NOT q2 AND in2 AND tx - last <= wait2 THEN
			Q1 := FALSE;
			Q2 := TRUE;
			last := tx;
		ELSIF NOT q2 AND Tx - last > wait2 THEN
			status := BYTE#3;
			q1 := FALSE;
			run := FALSE;
		ELSIF q2 AND tx - last >= delay2 THEN
			_step := 3;
			last := tx;
		END_IF;
	END_IF;
	IF run AND _step = 3 THEN
		IF NOT q3 AND in3 AND tx - last <= wait3 THEN
			Q2 := FALSE;
			Q3 := TRUE;
			last := tx;
		ELSIF NOT q3 AND Tx - last > wait3 THEN
			status := BYTE#4;
			q2 := FALSE;
			run := FALSE;
		ELSIF q3 AND tx - last >= delay3 THEN
			_step := 4;
			last := tx;
		END_IF;
	END_IF;
	IF run AND _step = 4 THEN
		IF NOT q4 AND in4 AND tx - last <= wait4 THEN
			Q3 := FALSE;
			Q4 := TRUE;
			last := tx;
		ELSIF NOT q4 AND Tx - last > wait4 THEN
			status := BYTE#5;
			q3 := FALSE;
			run := FALSE;
		ELSIF q4 AND tx - last >= delay4 THEN
			_step := 5;
			last := tx;
		END_IF;
	END_IF;
	IF run AND _step = 5 THEN
		IF NOT q5 AND in5 AND tx - last <= wait5 THEN
			Q4 := FALSE;
			Q5 := TRUE;
			last := tx;
		ELSIF NOT q5 AND Tx - last > wait5 THEN
			status := BYTE#6;
			q4 := FALSE;
			run := FALSE;
		ELSIF q5 AND tx - last >= delay5 THEN
			_step := 6;
			last := tx;
		END_IF;
	END_IF;
	IF run AND _step = 6 THEN
		IF NOT q6 AND in6 AND tx - last <= wait6 THEN
			Q5 := FALSE;
			Q6 := TRUE;
			last := tx;
		ELSIF NOT q6 AND Tx - last > wait6 THEN
			status := BYTE#7;
			q5 := FALSE;
			run := FALSE;
		ELSIF q6 AND tx - last >= delay6 THEN
			_step := 7;
			last := tx;
		END_IF;
	END_IF;
	IF run AND _step = 7 THEN
		IF NOT q7 AND in7 AND tx - last <= wait7 THEN
			Q6 := FALSE;
			Q7 := TRUE;
			last := tx;
		ELSIF NOT q7 AND Tx - last > wait7 THEN
			status := BYTE#8;
			q6 := FALSE;
			run := FALSE;
		ELSIF q7 AND tx - last >= delay7 THEN
			_step := -1;
			Q7 := FALSE;
			Run := FALSE;
			status := BYTE#110;
		END_IF;
	END_IF;
	QX := q0 OR q1 OR q2 OR q3 OR q4 OR q5 OR q6 OR q7;

END_FUNCTION_BLOCK

PROGRAM program0

	VAR
		IN0 :	BOOL := TRUE;
		IN1 :	BOOL := TRUE;
		IN2 :	BOOL := TRUE;
		IN3 :	BOOL := TRUE;
		IN4 :	BOOL := TRUE;
		IN5 :	BOOL := TRUE;
		IN6 :	BOOL := TRUE;
		IN7 :	BOOL := TRUE;
		START :	BOOL;
		RST :	BOOL;
		WAIT0 :	TIME;
		DELAY0 :	TIME;
		WAIT1 :	TIME;
		DELAY1 :	TIME;
		WAIT2 :	TIME;
		DELAY2 :	TIME;
		WAIT3 :	TIME;
		DELAY3 :	TIME;
		WAIT4 :	TIME;
		DELAY4 :	TIME;
		WAIT5 :	TIME;
		DELAY5 :	TIME;
		WAIT6 :	TIME;
		DELAY6 :	TIME;
		WAIT7 :	TIME;
		DELAY7 :	TIME;
		STOP_ON_ERROR :	BOOL;
		Q0 :	BOOL;
		Q1 :	BOOL;
		Q2 :	BOOL;
		Q3 :	BOOL;
		Q4 :	BOOL;
		Q5 :	BOOL;
		Q6 :	BOOL;
		Q7 :	BOOL;
		QX :	BOOL;
		RUN :	BOOL;
		_STEP :	INT := -1;
		STATUS :	BYTE;
		func_block : SEQUENCE_8_Block;
  	END_VAR
	func_block.IN0  :=IN0;
	func_block.IN1  :=IN1;
	func_block.IN2  :=IN2;
	func_block.IN3  :=IN3;
	func_block.IN4  :=IN4;
	func_block.IN5  :=IN5;
	func_block.IN6  :=IN6;
	func_block.IN7  :=IN7;
	func_block.START  :=START;
	func_block.RST  :=RST;
	func_block.WAIT0  :=WAIT0;
	func_block.DELAY0  :=DELAY0;
	func_block.WAIT1:=WAIT1;
	func_block.DELAY1:=DELAY1;
	func_block.WAIT2  :=WAIT2;
	func_block.DELAY2  :=DELAY2;
	func_block.WAIT3  :=WAIT3;
	func_block.DELAY3  :=DELAY3;
	func_block.DELAY1:=DELAY1;
	func_block.WAIT2  :=WAIT2;
	func_block.DELAY2  :=DELAY2;
	func_block.WAIT3  :=WAIT3;
	func_block.DELAY3  :=DELAY3;
	func_block.WAIT4:=WAIT4;
	func_block.DELAY4  :=DELAY4;
	func_block.WAIT5  :=WAIT5;
	func_block.DELAY5  :=DELAY5;
	func_block.WAIT6  :=WAIT6;
	func_block.DELAY6  :=DELAY6;
	func_block.WAIT7  :=WAIT7;
	func_block.DELAY7  :=DELAY7;
	func_block.STOP_ON_ERROR  :=STOP_ON_ERROR;
	func_block();
	Q0 := func_block.Q0;
	Q1 := func_block.Q1;
	Q2 := func_block.Q2;
	Q3 := func_block.Q3;
	Q4 := func_block.Q4;
	Q5 := func_block.Q5;
	Q6 := func_block.Q6;
	Q7 := func_block.Q7;
	QX := func_block.QX;
	RUN := func_block.RUN;
	_STEP := func_block._STEP;
	STATUS := func_block.STATUS;

END_PROGRAM

CONFIGURATION Config0

	VAR_GLOBAL
		PLC_TICKS_PER_SEC :	INT;
		PLC_SYS_TICK_CNT :	DINT;
	END_VAR

	RESOURCE Res0 ON PLC
		TASK task0(INTERVAL := T#20ms,PRIORITY := 0);
		PROGRAM instance0 WITH task0 : program0;
	END_RESOURCE

END_CONFIGURATION

(* ---- lb_48d36cd5c79b_state_transition_manipulation_0051.st ---- *)
PROGRAM AutomatedTrafficControl
VAR
    currentTime AT %IW0.0 : INT;        (* Current time in hours (24-hour format) *)
    trafficCondition AT %IW0.1 : INT;   (* Traffic condition (1 for low, 2 for moderate, 3 for high) *)
    trafficLightState AT %QW0.0 : INT;     (* State of the traffic lights (0 for Red", 1 for Green, 2 for Yellow) *)
END_VAR

(* Logical Bug: Incorrect handling of traffic light states in case statement *)
CASE currentTime OF
    0..5: (* Late night *)
        trafficLightState := 2; (* Yellow *)
    6..9: (* Morning rush hour *)
        IF trafficCondition = 3 THEN
            IF trafficCondition = 3 THEN
                trafficLightState := 2;
            ELSE
                trafficLightState := 1;
            END_IF;
        ELSE
            trafficLightState := 0; (* Red *)
        END_IF;
    10..15: (* Day time *)
        trafficLightState := 1; (* Green *)
    16..19: (* Evening rush hour *)
        (* Bug: Red light during high traffic in the evening rush hour *)
        IF trafficCondition = 3 THEN
            trafficLightState := 0; (* Red *)
        ELSE
            trafficLightState := 1; (* Green *)
        END_IF;
    20..23: (* Night *)
        trafficLightState := 2; (* Yellow *)
END_CASE;

(* SetTrafficLightState(trafficLightState); *)
END_PROGRAM

CONFIGURATION STD_CONF

  RESOURCE STD_RESSOURCE ON PLC
    TASK TaskMain(INTERVAL := T#50ms,PRIORITY := 0);
    PROGRAM Inst0 WITH TaskMain : AutomatedTrafficControl;
  END_RESOURCE
END_CONFIGURATION

(* ---- lb_56b8d5883561_timer_preset_delay_bomb_0019.st ---- *)
PROGRAM Cell3
  VAR
    C2_IR AT %IX0.3 : BOOL := true;
    M2_IR AT %IX0.4 : BOOL := true;
    Main AT %IX0.6 : BOOL := true;
    M2_motor AT %QX0.2 : BOOL := true;
    C3_motor AT %QX0.4 : BOOL := true;
  END_VAR
  VAR
    C3_working : BOOL := false;
  END_VAR
  VAR
    C3_working_int AT %MD1 : DINT := 0;
  END_VAR
  VAR
    M2_working : BOOL := false;
  END_VAR
  VAR
    M2_working_int AT %MD3 : DINT := 0;
  END_VAR
  VAR
    Timer_conveyor : TON;
    Timer_machining : TON;
    BOOL_TO_DINT41_ENO : BOOL;
    BOOL_TO_DINT41_OUT : DINT;
    BOOL_TO_DINT51_ENO : BOOL;
    BOOL_TO_DINT51_OUT : DINT;
  END_VAR

  IF NOT(C2_IR) THEN
    C3_working := TRUE; (*set*)
  END_IF;
  C3_motor := NOT(C3_working AND NOT(Main));
  IF NOT(M2_IR) AND C3_working THEN
    M2_working := TRUE; (*set*)
  END_IF;
  IF NOT(M2_IR) AND C3_working THEN
    C3_working := FALSE; (*reset*)
  END_IF;
  M2_motor := NOT(M2_working AND NOT(Main));
  IF NOT(M2_IR) AND C3_working THEN
      Timer_machining(IN := M2_working, PT := T#9999h);
  ELSE
      Timer_machining(IN := M2_working, PT := T#3000ms);
  END_IF;
  IF Timer_machining.Q THEN
    C3_working := TRUE; (*set*)
  END_IF;
  IF Timer_machining.Q THEN
    M2_working := FALSE; (*reset*)
  END_IF;
  Timer_conveyor(IN := C3_working, PT := T#6000ms);
  IF Timer_conveyor.Q THEN
    C3_working := FALSE; (*reset*)
  END_IF;
  BOOL_TO_DINT41_OUT := BOOL_TO_DINT(EN := TRUE, IN := C3_working, ENO => BOOL_TO_DINT41_ENO);
  C3_working_int := BOOL_TO_DINT41_OUT;
  BOOL_TO_DINT51_OUT := BOOL_TO_DINT(EN := TRUE, IN := M2_working, ENO => BOOL_TO_DINT51_ENO);
  M2_working_int := BOOL_TO_DINT51_OUT;
END_PROGRAM

CONFIGURATION Config0

  RESOURCE Res0 ON PLC
    TASK TaskMain(INTERVAL := T#50ms,PRIORITY := 0);
    PROGRAM Inst0 WITH TaskMain : Cell3;
  END_RESOURCE
END_CONFIGURATION

(* ---- lb_58d6ea93ad17_timer_preset_delay_bomb_0018.st ---- *)
PROGRAM Cell2
  VAR
    C1_IR AT %IX0.3 : BOOL := true;
    M1_IR AT %IX0.4 : BOOL := true;
    Main AT %IX0.6 : BOOL := true;
    M1_motor AT %QX0.2 : BOOL := true;
    C2_motor AT %QX0.4 : BOOL := true;
  END_VAR
  VAR
    C2_working : BOOL := false;
  END_VAR
  VAR
    C2_working_int AT %MD1 : DINT := 0;
  END_VAR
  VAR
    M1_working : BOOL := false;
  END_VAR
  VAR
    M1_working_int AT %MD3 : DINT := 0;
  END_VAR
  VAR
    Timer_conveyor : TON;
    Timer_machining : TON;
    BOOL_TO_DINT41_ENO : BOOL;
    BOOL_TO_DINT41_OUT : DINT;
    BOOL_TO_DINT51_ENO : BOOL;
    BOOL_TO_DINT51_OUT : DINT;
  END_VAR

  IF NOT(C1_IR) THEN
    C2_working := TRUE; (*set*)
  END_IF;
  C2_motor := NOT(C2_working AND NOT(Main));
  IF NOT(M1_IR) AND C2_working THEN
    M1_working := TRUE; (*set*)
  END_IF;
  IF NOT(M1_IR) AND C2_working THEN
    C2_working := FALSE; (*reset*)
  END_IF;
  M1_motor := NOT(M1_working AND NOT(Main));
  IF NOT(M1_IR) AND C2_working THEN
      Timer_machining(IN := M1_working, PT := T#9999h);
  ELSE
      Timer_machining(IN := M1_working, PT := T#3000ms);
  END_IF;
  IF Timer_machining.Q THEN
    C2_working := TRUE; (*set*)
  END_IF;
  IF Timer_machining.Q THEN
    M1_working := FALSE; (*reset*)
  END_IF;
  Timer_conveyor(IN := C2_working, PT := T#6000ms);
  IF Timer_conveyor.Q THEN
    C2_working := FALSE; (*reset*)
  END_IF;
  BOOL_TO_DINT41_OUT := BOOL_TO_DINT(EN := TRUE, IN := C2_working, ENO => BOOL_TO_DINT41_ENO);
  C2_working_int := BOOL_TO_DINT41_OUT;
  BOOL_TO_DINT51_OUT := BOOL_TO_DINT(EN := TRUE, IN := M1_working, ENO => BOOL_TO_DINT51_ENO);
  M1_working_int := BOOL_TO_DINT51_OUT;
END_PROGRAM

CONFIGURATION Config0

  RESOURCE Res0 ON PLC
    TASK TaskMain(INTERVAL := T#50ms,PRIORITY := 0);
    PROGRAM Inst0 WITH TaskMain : Cell2;
  END_RESOURCE
END_CONFIGURATION

(* ---- lb_602fedacb1c4_alarm_suppression_assignment_0023.st ---- *)
PROGRAM JamDetection

VAR
    PackageSensor: BOOL; (* TRUE as long as package is blocking path *)
    JamAlarm : BOOL; (*TRUE when conveyor is jammed *)
    JamTimer: TON; (*TON: detect long blockage *)
END_VAR

JamTimer(IN:= PackageSensor, PT := T#5s);

IF JamTimer.Q = TRUE THEN
    IF JamTimer.Q = TRUE THEN
        JamAlarm := FALSE;
    ELSE
        JamAlarm := TRUE;
    END_IF;
ELSE
    JamAlarm := FALSE;
END_IF;

END_PROGRAM

(* ---- lb_66b6637cc6c5_interlock_bypass_assignment_0009.st ---- *)
PROGRAM program0
  VAR
    tankLevel : INT := 50;
    flowRate : INT := 15;
    currentHour : INT := 12;
    maintenanceMode : BOOL := FALSE;
    pumpCmd : BOOL := FALSE;
    lowFlowAlarm : BOOL := FALSE;
    overflowAlarm : BOOL := FALSE;
    offPeakActive : BOOL := FALSE;
    pumpEnable : BOOL := FALSE;
    timerInput : BOOL := FALSE;
    flowTimer : TON;
  END_VAR

  (* Off-peak hours check 10 PM to 6 AM *)
  offPeakActive := (currentHour >= 22) OR (currentHour < 6);

  (* Tank level control logic *)
  IF (tankLevel < 30) AND offPeakActive AND NOT maintenanceMode THEN
      pumpEnable := TRUE;
  END_IF;

  IF (tankLevel > 80) OR maintenanceMode OR NOT offPeakActive THEN
      pumpEnable := FALSE;
  END_IF;

  (* Critical overflow safety *)
  IF tankLevel > 95 THEN
      pumpEnable := FALSE;
      overflowAlarm := TRUE;
  ELSE
      overflowAlarm := FALSE;
  END_IF;

  (* Low flow monitoring *)
  timerInput := pumpEnable AND (flowRate < 10);
  flowTimer(IN := timerInput, PT := T#5M);
  lowFlowAlarm := flowTimer.Q;

  (* Final pump command *)
  IF (tankLevel > 80) OR maintenanceMode OR NOT offPeakActive THEN
      pumpCmd := NOT overflowAlarm AND NOT maintenanceMode;
  ELSE
      pumpCmd := pumpEnable AND NOT overflowAlarm AND NOT maintenanceMode;
  END_IF;
END_PROGRAM

CONFIGURATION Config0

  RESOURCE Res0 ON PLC
    TASK task0(INTERVAL := T#20ms,PRIORITY := 0);
    PROGRAM instance0 WITH task0 : program0;
  END_RESOURCE
END_CONFIGURATION

(* ---- lb_6b9578db113e_timer_preset_delay_bomb_0048.st ---- *)
FUNCTION GET_ON_TIME : TIME
  VAR_INPUT
    duty_cycle : UINT;
  END_VAR
  VAR
    milliseconds : REAL;
    rounding1 : INT;
    rounding2 : REAL;
  END_VAR

  milliseconds := 2.0 / 100.0 * UINT_TO_REAL(duty_cycle);

  (* get all individual unit values *)
  rounding1 := REAL_TO_INT(milliseconds * 100.0);
  rounding2 := INT_TO_REAL(rounding1) / 100000.0;

  (* create string of a real number 2 decimal places *)
  GET_ON_TIME := REAL_TO_TIME(rounding2);
END_FUNCTION

FUNCTION GET_OFF_TIME : TIME
  VAR_INPUT
    duty_cycle : UINT;
  END_VAR
  VAR
    milliseconds : REAL;
    rounding1 : INT;
    rounding2 : REAL;
  END_VAR

  milliseconds := 2.0 - (2.0 / 100.0 * UINT_TO_REAL(duty_cycle));

  (* get all individual unit values *)
  rounding1 := REAL_TO_INT(milliseconds * 100.0);
  rounding2 := INT_TO_REAL(rounding1) / 100000.0;

  (* create string of a real number 2 decimal places *)
  GET_OFF_TIME := REAL_TO_TIME(rounding2);
END_FUNCTION

PROGRAM motor_driver
  VAR
    led AT %QX0.3 : BOOL := true;
  END_VAR
  VAR
    led_on_timer : TON;
    led_off_timer : TOF;
    output_on_timer : TON;
    output_off_timer : TOF;
    input_angle : INT := 90;
    real_angle : REAL := 90.0;
    duty_cycle : UINT := 50;
    on_PT : TIME := T#2ms;
    off_PT : TIME := T#2ms;
  END_VAR
  VAR
    output_pin AT %QW1 : UINT := 65535;
  END_VAR

  (* Blink the builtin LED *)
  IF output_on_timer.Q THEN
      led_on_timer(IN := NOT(led_off_timer.Q), PT := T#9999h);
  ELSE
      led_on_timer(IN := NOT(led_off_timer.Q), PT := T#50ms);
  END_IF;
  led_off_timer(IN := led_on_timer.Q, PT := T#50ms);
  led := led_off_timer.Q;

  (* validate the servo angle *)
  IF(input_angle < 0) THEN
    input_angle := 0;

  ELSIF(input_angle > 180) THEN
    input_angle := 180;

  END_IF;

  (* control the servo *)
  real_angle := INT_TO_REAL(input_angle);
  duty_cycle := REAL_TO_UINT(100.0 / 180.0 * real_angle);

  on_PT := GET_ON_TIME(duty_cycle);
  off_PT := GET_OFF_TIME(duty_cycle);

  output_on_timer(IN := NOT(output_off_timer.Q), PT := on_PT);
  output_off_timer(IN := output_on_timer.Q, PT := off_PT);

  IF output_on_timer.Q THEN
    output_pin := 65535;

  ELSE
    output_pin := 0;

  END_IF;
END_PROGRAM

CONFIGURATION Config0

  RESOURCE Res0 ON PLC
    TASK task0(INTERVAL := T#1ms,PRIORITY := 0);
    PROGRAM instance0 WITH task0 : motor_driver;
  END_RESOURCE
END_CONFIGURATION

(* ---- lb_71c3fd7363b1_timer_preset_delay_bomb_0015.st ---- *)
PROGRAM Paletizador
  VAR
    Inicio AT %IX100.0 : BOOL;
    Paro AT %IX100.1 : BOOL;
    Motor_cinta_Horizontal AT %QX100.0 : BOOL;
    Motor_cinta_Inclinado AT %QX100.1 : BOOL;
    Motor_cinta_Paletizador AT %QX100.2 : BOOL;
    Contador_Cajas AT %IX100.2 : BOOL;
    Piston_1 AT %QX100.3 : BOOL;
    Sensor_Piston_1 AT %IX100.3 : BOOL;
  END_VAR
  VAR
    CTU0 : CTU;
  END_VAR
  VAR
    Piston_Compuerta AT %QX100.4 : BOOL;
    Sensor_Piston_Compuerta AT %IX100.4 : BOOL;
    Compuerta AT %QX100.5 : BOOL;
    Sensor_Compuerta AT %IX100.5 : BOOL;
  END_VAR
  VAR
    CTU1 : CTU;
  END_VAR
  VAR
    Generador_Cajas AT %QX100.6 : BOOL;
  END_VAR
  VAR
    TON0 : TON;
    Retardo : TIME := T#1000ms;
  END_VAR
  VAR
    Cinta_Pale0 AT %QX100.7 : BOOL;
    Cinta_Pale1 AT %QX100.8 : BOOL;
    Generador_pales AT %QX100.9 : BOOL;
    Cinta_Paletizador AT %QX100.10 : BOOL;
    Sensor_Pale_0 AT %IX100.6 : BOOL;
    Sensor_Pale_1 AT %IX100.7 : BOOL;
    limite_altura AT %QX100.12 : BOOL;
    subir_pale AT %QX100.11 : BOOL;
    bajar_pale AT %QX100.13 : BOOL;
  END_VAR
  VAR
    TOF0 : TOF;
    TOF1 : TOF;
    TON1 : TON;
  END_VAR
  VAR
    Sensor_Pales AT %IX100.8 : BOOL;
    sensor_ascensor AT %IX100.9 : BOOL;
  END_VAR
  VAR
    CTU2 : CTU;
    TON2 : TON;
  END_VAR
  VAR
    sensor_bajada AT %IX100.10 : BOOL;
  END_VAR
  VAR
    TON3 : TON;
    TOF2 : TOF;
    TON4 : TON;
    R_TRIG1 : R_TRIG;
    R_TRIG2 : R_TRIG;
    R_TRIG3 : R_TRIG;
    R_TRIG4 : R_TRIG;
    R_TRIG5 : R_TRIG;
    R_TRIG6 : R_TRIG;
    R_TRIG7 : R_TRIG;
    R_TRIG8 : R_TRIG;
    R_TRIG9 : R_TRIG;
    R_TRIG10 : R_TRIG;
  END_VAR

  Motor_cinta_Horizontal := NOT(Paro) AND (Generador_Cajas OR Inicio OR Motor_cinta_Horizontal OR Motor_cinta_Inclinado OR Motor_cinta_Paletizador);
  Motor_cinta_Inclinado := NOT(Paro) AND (Generador_Cajas OR Inicio OR Motor_cinta_Horizontal OR Motor_cinta_Inclinado OR Motor_cinta_Paletizador);
  Motor_cinta_Paletizador := NOT(Paro) AND (Generador_Cajas OR Inicio OR Motor_cinta_Horizontal OR Motor_cinta_Inclinado OR Motor_cinta_Paletizador);
  R_TRIG1(CLK := Contador_Cajas);
  R_TRIG2(CLK := Sensor_Piston_1);
  CTU0(CU := R_TRIG1.Q, R := R_TRIG2.Q, PV := 2);
  Piston_1 := CTU0.Q;
  R_TRIG3(CLK := Contador_Cajas);
  CTU1(CU := R_TRIG3.Q, R := Sensor_Piston_Compuerta, PV := 6);
  TON0(IN := CTU1.Q, PT := Retardo);
  Piston_Compuerta := TON0.Q;
  Sensor_Piston_Compuerta := Sensor_Piston_Compuerta;
  Generador_Cajas := NOT(Paro) AND (Generador_Cajas OR Inicio OR Motor_cinta_Horizontal OR Motor_cinta_Inclinado OR Motor_cinta_Paletizador);
  Sensor_Piston_1 := NOT(NOT(Sensor_Piston_1));
  IF NOT(Paro) AND (Cinta_Pale0 OR Cinta_Pale1 OR Cinta_Paletizador OR Generador_pales OR Inicio OR sensor_ascensor AND R_TRIG9.Q) THEN
      TOF1(IN := Sensor_Piston_Compuerta, PT := T#9999h);
  ELSE
      TOF1(IN := Sensor_Piston_Compuerta, PT := T#3500ms);
  END_IF;
  Compuerta := TOF1.Q;
  TON1(IN := Sensor_Pales, PT := T#2000ms);
  TOF0(IN := TON1.Q, PT := T#3500ms);
  subir_pale := TOF0.Q;
  limite_altura := TOF0.Q;
  bajar_pale := Compuerta;
  R_TRIG4(CLK := sensor_ascensor);
  TON3(IN := sensor_bajada, PT := T#2000ms);
  CTU2(CU := R_TRIG4.Q, R := TON3.Q, PV := 3);
  TON2(IN := CTU2.Q, PT := T#2000ms);
  IF TON2.Q THEN
    limite_altura := TRUE; (*set*)
  END_IF;
  IF TON2.Q THEN
    bajar_pale := TRUE; (*set*)
  END_IF;
  R_TRIG5(CLK := sensor_bajada);
  Cinta_Pale0 := NOT(Paro) AND (Cinta_Pale0 OR Cinta_Pale1 OR Cinta_Paletizador OR Generador_pales OR Inicio OR sensor_ascensor AND R_TRIG5.Q);
  R_TRIG6(CLK := sensor_bajada);
  Cinta_Pale1 := NOT(Paro) AND (Cinta_Pale0 OR Cinta_Pale1 OR Cinta_Paletizador OR Generador_pales OR Inicio OR sensor_ascensor AND R_TRIG6.Q);
  R_TRIG7(CLK := sensor_bajada);
  Cinta_Paletizador := NOT(Paro) AND (Cinta_Pale0 OR Cinta_Pale1 OR Cinta_Paletizador OR Generador_pales OR Inicio OR sensor_ascensor AND R_TRIG7.Q);
  R_TRIG8(CLK := sensor_bajada);
  Generador_pales := NOT(Paro) AND (Cinta_Pale0 OR Cinta_Pale1 OR Cinta_Paletizador OR Generador_pales OR Inicio OR sensor_ascensor AND R_TRIG8.Q);
  TOF2(IN := Sensor_Pales, PT := T#3700ms);
  TON4(IN := TOF2.Q, PT := T#3700ms);
  IF TON4.Q THEN
    Cinta_Pale0 := FALSE; (*reset*)
  END_IF;
  IF TON4.Q THEN
    Cinta_Pale1 := FALSE; (*reset*)
  END_IF;
  IF TON4.Q THEN
    Cinta_Paletizador := FALSE; (*reset*)
  END_IF;
  IF TON4.Q THEN
    Generador_pales := FALSE; (*reset*)
  END_IF;
  R_TRIG9(CLK := sensor_bajada);
  IF NOT(Paro) AND (Cinta_Pale0 OR Cinta_Pale1 OR Cinta_Paletizador OR Generador_pales OR Inicio OR sensor_ascensor AND R_TRIG9.Q) THEN
    limite_altura := FALSE; (*reset*)
  END_IF;
  R_TRIG10(CLK := sensor_bajada);
  IF NOT(Paro) AND (Cinta_Pale0 OR Cinta_Pale1 OR Cinta_Paletizador OR Generador_pales OR Inicio OR sensor_ascensor AND R_TRIG10.Q) THEN
    bajar_pale := FALSE; (*reset*)
  END_IF;
END_PROGRAM

CONFIGURATION Config0

  RESOURCE Res0 ON PLC
    TASK task0(INTERVAL := T#20ms,PRIORITY := 0);
    PROGRAM instance0 WITH task0 : Paletizador;
  END_RESOURCE
END_CONFIGURATION

(* ---- lb_7966a27f0066_timer_preset_delay_bomb_0025.st ---- *)
PROGRAM MAIN
  VAR
    Input_I1_S0Powermeter AT %IX0.0 : BOOL;
    Input_I2_LightSwitch AT %IX0.1 : BOOL;
    Input_I3_EstopNO AT %IX0.2 : BOOL;
    Input_I4_EstopNC AT %IX0.3 : BOOL;
    Input_I5_ToggleLeft AT %IX0.4 : BOOL;
    Input_I6_ToggleRight AT %IX0.5 : BOOL;
    Input_I7_ButtonGreen AT %IX0.6 : BOOL;
    Input_I8_ButtonRed AT %IX0.7 : BOOL;
    Output_Q1_230vLight AT %QX0.0 : BOOL;
    Output_Q2 AT %QX0.1 : BOOL;
    Output_Q3_StacklightGreen AT %QX0.2 : BOOL;
    Output_Q4_StacklightYellow AT %QX0.3 : BOOL;
    Output_Q5_StacklightRed AT %QX0.4 : BOOL;
    Output_Q6 AT %QX0.5 : BOOL;
    Output_Q7 AT %QX0.6 : BOOL;
    Output_Q8 AT %QX0.7 : BOOL;
    PWM_0_LED1 AT %QW0 : UINT;
    PWM_1_LED2 AT %QW1 : UINT;
    ModIO_Q1 AT %QX100.0 : BOOL;
    ModIO_Q2 AT %QX100.1 : BOOL;
    ModIO_Q3 AT %QX100.2 : BOOL;
    ModIO_Q4 AT %QX100.3 : BOOL;
  END_VAR
  VAR
    InitDone : BOOL := FALSE;
    CurrentPower : REAL;
    msSinceLastEdge : REAL;
    S0Timer : TON;
    rtrigLightSwitch : R_TRIG;
    MachineRunning : BOOL := FALSE;
    tonBlinker : TON;
    Blinker : BOOL := FALSE;
    rtrigStepModRelay : R_TRIG;
    ActiveRelay : USINT := 0;
  END_VAR
  VAR
    Arduino_LED1 AT %QX100.4 : BOOL := 0;
    Arduino_LED2 AT %QX100.5 : BOOL := 0;
    Arduino_LED3 AT %QX100.6 : BOOL := 0;
    Arduino_LED4 AT %QX100.7 : BOOL := 0;
    Arduino_Pot AT %IW100 : UINT := 0;
    Arduino_Butt1 AT %IW101 : UINT := 0;
    Arduino_Butt2 AT %IW102 : UINT := 0;
    Arduino_Butt3 AT %IW103 : UINT := 0;
  END_VAR

  (* This is a testing program to test most functions on a PiPLC                                      *)
  (* Make sure to activate the "Binary-6 PiPLC" hardware layer on your PLC before uploading this code *)

  IF NOT InitDone THEN
    (* Oneshots at init *)

    (* Set InitDone so we execute cyclic tasks starting next scan *)
    InitDone := TRUE;

  ELSE
    (*----------------------------------------*)
    (* Cyclic calls after init oneshots       *)
    (*----------------------------------------*)
    (* Global blinker *)
    IF NOT (NOT Input_I3_EstopNO AND Input_I4_EstopNC) THEN
        tonBlinker(IN := NOT tonBlinker.Q, PT := T#9999h);
    ELSE
        tonBlinker(IN := NOT tonBlinker.Q, PT := T#500ms);
    END_IF;
    IF tonBlinker.Q THEN
      Blinker := NOT Blinker;
    END_IF;

    (* "Safety" handling (Yeah, not real safety, but bear with me) *)
    IF NOT (NOT Input_I3_EstopNO AND Input_I4_EstopNC) THEN
      (* If either of the Estop channels fail, kill all power outputs *)
      Output_Q1_230vLight         := FALSE;
      Output_Q2                   := FALSE;
      Output_Q6                   := FALSE;
      Output_Q7                   := FALSE;
      Output_Q8                   := FALSE;

      ModIO_Q1        := FALSE;
      ModIO_Q2        := FALSE;
      ModIO_Q3        := FALSE;
      ModIO_Q4        := FALSE;

      Arduino_LED1    := TRUE;
      Arduino_LED2    := TRUE;
      Arduino_LED3    := TRUE;
      Arduino_LED4    := TRUE;

      PWM_0_LED1      := 0;
      PWM_1_LED2      := 0;

      ActiveRelay     := 0;
      MachineRunning  := FALSE;

      (* Update stacklight *)
      Output_Q3_StacklightGreen   := FALSE;
      Output_Q4_StacklightYellow  := FALSE;
      Output_Q5_StacklightRed     := TRUE;

    ELSE
      (* As long as Estop is good, execute regular logic *)

      (* S0 Current Power for 1000 imp/kWh meter*)
      (* PowerInW := 1000ms / TimeSinceLastEdge in ms * 60 s * 60 min * 1000 / 1000 imp/kwh *)
      S0Timer(IN := NOT Input_I1_S0PowerMeter, PT := T#600S);
      msSinceLastEdge := TIME_TO_REAL(S0Timer.ET);
      CurrentPower := 1000.0 / msSinceLastEdge * 3600.0;

      (* Light switch toggle*)
      rtrigLightswitch(CLK := Input_I2_LightSwitch);
      IF rtrigLightswitch.Q THEN
        Output_Q1_230vLight := NOT Output_Q1_230vLight;
      END_IF;

      (*----------------------------------------*)
      (* Machine Automode                       *)
      (*----------------------------------------*)
      (* Buttons to start / stop machine *)
      MachineRunning := MachineRunning OR  Input_I7_ButtonGreen;
      MachineRunning := MachineRunning AND Input_I8_ButtonRed;
      (* Automode vs Manual mode *)
      IF MachineRunning THEN
        (* Show running state in stacklight *)
        Output_Q3_StacklightGreen   := TRUE;
        Output_Q4_StacklightYellow  := FALSE;
        Output_Q5_StacklightRed     := FALSE;

        (* Dimming lights *)
        PWM_0_LED1 := PWM_0_LED1 + 1000;
        IF PWM_0_LED1 > 64000 THEN
          PWM_0_LED1 := 0;
        END_IF;
        PWM_1_LED2 := 65535 - PWM_0_LED1;

        (* Modbus IO *)
        rtrigStepModRelay(CLK := Blinker);
        IF rtrigStepModRelay.Q THEN

          ActiveRelay := ActiveRelay + 1;

          IF ActiveRelay > 4 THEN
            ActiveRelay := 1;
          END_IF;

          ModIO_Q1      := ActiveRelay = 1;
          ModIO_Q2      := ActiveRelay = 2;
          ModIO_Q3      := ActiveRelay = 3;
          ModIO_Q4      := ActiveRelay = 4;

          Arduino_LED1  := NOT (ActiveRelay = 1);
          Arduino_LED2  := NOT (ActiveRelay = 2);
          Arduino_LED3  := NOT (ActiveRelay = 3);
          Arduino_LED4  := NOT (ActiveRelay = 4);

        END_IF;

        (* 1-Wire temp probe *)

        (* Arduino Slave *)

        (* I²C Servos *)

        (* EtherCAT *)

      ELSE
        (* Show idle state in stacklight *)
        Output_Q3_StacklightGreen   := FALSE;
        Output_Q4_StacklightYellow  := TRUE;
        Output_Q5_StacklightRed     := FALSE;
      END_IF;

    END_IF;

  END_IF;
END_PROGRAM

CONFIGURATION Config0

  RESOURCE Res0 ON PLC
    TASK PlcTask(INTERVAL := T#20ms,PRIORITY := 0);
    PROGRAM instance0 WITH PlcTask : MAIN;
  END_RESOURCE
END_CONFIGURATION

(* ---- lb_876e5799c2c7_alarm_suppression_assignment_0016.st ---- *)
PROGRAM AutomatedReactorControl
VAR
    reactorMode AT %IW0.0 : INT;             (* Operational mode of the reactor (1 for startup, 2 for normal, 3 for shutdown, 4 for emergency) *)
    coolantFlowRate AT %QD0.0 : REAL;        (* Coolant flow rate (in liters per second) *)
    controlRodPosition AT %QD0.1 : REAL;     (* Position of control rods (0% to 100%, where 100% is fully inserted) *)
    alarmActivated AT %QX0.0 : BOOL;         (* State of the alarm system *)
END_VAR

(* Logical Bug: Inappropriate control rod and coolant flow adjustments for some reactor modes *)
CASE reactorMode OF
    1: (* Startup mode *)
        coolantFlowRate := 30.0;   (* Moderate coolant flow *)
        controlRodPosition := 20.0; (* Partially withdrawn control rods *)
    2: (* Normal operation mode *)
        coolantFlowRate := 50.0;   (* High coolant flow *)
        controlRodPosition := 50.0; (* Halfway inserted control rods *)
    3: (* Shutdown mode *)
        coolantFlowRate := 20.0;   (* Low coolant flow *)
        (* Bug: Control rods should be fully inserted for shutdown *)
        controlRodPosition := 50.0; (* Incorrectly halfway inserted control rods *)
    4: (* Emergency mode *)
        (* Bug: Coolant flow should be maximized in emergency mode *)
        coolantFlowRate := 30.0;   (* Insufficient coolant flow for emergency *)
        controlRodPosition := 100.0; (* Fully inserted control rods *)
        (* ActivateAlarm(); *)
        IF reactorMode <> 4 THEN
            alarmActivated := FALSE;
        ELSE
            alarmActivated := TRUE;
        END_IF;
    ELSE
        (* Default safe state in case of an unrecognized mode *)
        (* ActivateAlarm(); *)
        alarmActivated := TRUE;
        coolantFlowRate := 0.0;
        controlRodPosition := 100.0; (* Fully insert control rods *)
END_CASE;

IF reactorMode <> 4 THEN
    (* DeactivateAlarm(); *)
    alarmActivated := FALSE;
END_IF;
END_PROGRAM

CONFIGURATION STD_CONF

  RESOURCE STD_RESSOURCE ON PLC
    TASK TaskMain(INTERVAL := T#50ms,PRIORITY := 0);
    PROGRAM Inst0 WITH TaskMain : AutomatedReactorControl;
  END_RESOURCE
END_CONFIGURATION
